LIN {X 0,Y 168.343,Z 1185.005,A -85,B 0,C 180,E1 2241.805,E2 2241.805} C_VEL
LIN {X 0,Y 169.597,Z 1183.384,A -85,B 0,C 180,E1 2234.616,E2 2234.616} C_VEL
LIN {X 0,Y 172.473,Z 1180.747,A -85,B 0,C 180,E1 2227.505,E2 2227.505} C_VEL
LIN {X 0,Y 177.252,Z 1177.063,A -85,B 0,C 180,E1 2220.61,E2 2220.61} C_VEL
LIN {X 0,Y 185.536,Z 1171.322,A -85,B 0,C 180,E1 2212.874,E2 2212.874} C_VEL
LIN {X 0,Y 197.006,Z 1163.471,A -85,B 0,C 180,E1 2205.542,E2 2205.542} C_VEL
LIN {X 0,Y 208.194,Z 1155.807,A -85,B 0,C 180,E1 2200.217,E2 2200.217} C_VEL
LIN {X 0,Y 221.519,Z 1146.423,A -85,B 0,C 180,E1 2195.217,E2 2195.217} C_VEL
LIN {X 0,Y 239.062,Z 1133.277,A -85,B 0,C 180,E1 2190.029,E2 2190.029} C_VEL
LIN {X 0,Y 253.681,Z 1121.544,A -85,B 0,C 180,E1 2186.529,E2 2186.529} C_VEL
LIN {X 0,Y 268.978,Z 1108.424,A -85,B 0,C 180,E1 2183.438,E2 2183.438} C_VEL
LIN {X 0,Y 287.731,Z 1090.816,A -85,B 0,C 180,E1 2180.24,E2 2180.24} C_VEL
LIN {X 0,Y 302.104,Z 1076.015,A -85,B 0,C 180,E1 2178.127,E2 2178.127} C_VEL
LIN {X 0,Y 316.159,Z 1060.322,A -85,B 0,C 180,E1 2176.294,E2 2176.294} C_VEL
LIN {X 0,Y 332.424,Z 1040.407,A -85,B 0,C 180,E1 2174.415,E2 2174.415} C_VEL
LIN {X 0,Y 346.747,Z 1020.63,A -85,B 0,C 180,E1 2172.929,E2 2172.929} C_VEL
LIN {X 0,Y 358.555,Z 1002.66,A -85,B 0,C 180,E1 2171.818,E2 2171.818} C_VEL
LIN {X 0,Y 370.024,Z 983.317,A -85,B 0,C 180,E1 2170.814,E2 2170.814} C_VEL
LIN {X 0,Y 383.165,Z 957.986,A -85,B 0,C 180,E1 2169.75,E2 2169.75} C_VEL
LIN {X 0,Y 392.344,Z 937.557,A -85,B 0,C 180,E1 2169.059,E2 2169.059} C_VEL
LIN {X 0,Y 400.34,Z 917.228,A -85,B 0,C 180,E1 2168.494,E2 2168.494} C_VEL
LIN {X 0,Y 408.607,Z 892.645,A -85,B 0,C 180,E1 2167.932,E2 2167.932} C_VEL
LIN {X 0,Y 415.555,Z 866.383,A -85,B 0,C 180,E1 2167.476,E2 2167.476} C_VEL
LIN {X 0,Y 420.191,Z 844.048,A -85,B 0,C 180,E1 2167.159,E2 2167.159} C_VEL
LIN {X 0,Y 424.177,Z 817.755,A -85,B 0,C 180,E1 2166.815,E2 2166.815} C_VEL
LIN {X 0,Y 442.106,Z 663.834,A -85,B 0,C 180,E1 2164.898,E2 2164.898} C_VEL
LIN {X 0,Y 441.771,Z 661.822,A -85,B 0,C 180,E1 2162.724,E2 2162.724} C_VEL
LIN {X 0,Y 442.134,Z 661.954,A -85,B 0,C 180,E1 2159.482,E2 2159.482} C_VEL
LIN {X 0,Y 442.426,Z 662.695,A -85,B 0,C 180,E1 2158.54,E2 2158.54} C_VEL
LIN {X 0,Y 440.538,Z 678.75,A -85,B 0,C 180,E1 2158.335,E2 2158.335} C_VEL
LIN {X 0,Y 439.566,Z 686.453,A -85,B 0,C 180,E1 2158.372,E2 2158.372} C_VEL
LIN {X 0,Y 436.764,Z 707.079,A -85,B 0,C 180,E1 2158.925,E2 2158.925} C_VEL
LIN {X 0,Y 435.94,Z 713.684,A -85,B 0,C 180,E1 2158.942,E2 2158.942} C_VEL
LIN {X 0,Y 422.165,Z 828.688,A -85,B 0,C 180,E1 2157.483,E2 2157.483} C_VEL
LIN {X 0,Y 417.336,Z 856.018,A -85,B 0,C 180,E1 2157.112,E2 2157.112} C_VEL
LIN {X 0,Y 411.12,Z 881.201,A -85,B 0,C 180,E1 2156.722,E2 2156.722} C_VEL
LIN {X 0,Y 404.786,Z 902.207,A -85,B 0,C 180,E1 2156.312,E2 2156.312} C_VEL
LIN {X 0,Y 397.021,Z 924.035,A -85,B 0,C 180,E1 2155.787,E2 2155.787} C_VEL
LIN {X 0,Y 385.817,Z 950.494,A -85,B 0,C 180,E1 2154.997,E2 2154.997} C_VEL
LIN {X 0,Y 375.845,Z 970.771,A -85,B 0,C 180,E1 2154.247,E2 2154.247} C_VEL
LIN {X 0,Y 364.942,Z 990.522,A -85,B 0,C 180,E1 2153.372,E2 2153.372} C_VEL
LIN {X 0,Y 350.842,Z 1013.342,A -85,B 0,C 180,E1 2152.137,E2 2152.137} C_VEL
LIN {X 0,Y 336.327,Z 1033.918,A -85,B 0,C 180,E1 2150.753,E2 2150.753} C_VEL
LIN {X 0,Y 323.015,Z 1051.093,A -85,B 0,C 180,E1 2149.357,E2 2149.357} C_VEL
LIN {X 0,Y 308.128,Z 1068.687,A -85,B 0,C 180,E1 2147.617,E2 2147.617} C_VEL
LIN {X 0,Y 289.64,Z 1088.449,A -85,B 0,C 180,E1 2145.148,E2 2145.148} C_VEL
LIN {X 0,Y 274.268,Z 1103.426,A -85,B 0,C 180,E1 2142.774,E2 2142.774} C_VEL
LIN {X 0,Y 259.412,Z 1116.892,A -85,B 0,C 180,E1 2140.13,E2 2140.13} C_VEL
LIN {X 0,Y 241.293,Z 1132.218,A -85,B 0,C 180,E1 2136.299,E2 2136.299} C_VEL
LIN {X 0,Y 224.396,Z 1145.324,A -85,B 0,C 180,E1 2131.915,E2 2131.915} C_VEL
LIN {X 0,Y 210.851,Z 1155.366,A -85,B 0,C 180,E1 2127.574,E2 2127.574} C_VEL
LIN {X 0,Y 197.418,Z 1165.01,A -85,B 0,C 180,E1 2122.194,E2 2122.194} C_VEL
LIN {X 0,Y 183.406,Z 1174.86,A -85,B 0,C 180,E1 2114.689,E2 2114.689} C_VEL
LIN {X 0,Y 174.298,Z 1181.394,A -85,B 0,C 180,E1 2107.865,E2 2107.865} C_VEL
LIN {X 0,Y 167.735,Z 1186.474,A -85,B 0,C 180,E1 2100.84,E2 2100.84} C_VEL
LIN {X 0,Y 163.294,Z 1190.442,A -85,B 0,C 180,E1 2093.453,E2 2093.453} C_VEL
LIN {X 0,Y 160.718,Z 1193.56,A -85,B 0,C 180,E1 2085.146,E2 2085.146} C_VEL
LIN {X 0,Y 160.036,Z 1195.327,A -85,B 0,C 180,E1 2077.177,E2 2077.177} C_VEL
LIN {X 0,Y 160.041,Z 1195.799,A -85,B 0,C 180,E1 2070.715,E2 2070.715} C_VEL
LIN {X 0,Y 160.019,Z 1195.475,A -85,B 0,C 180,E1 2064.621,E2 2064.621} C_VEL
LIN {X 0,Y 160.309,Z 1194.285,A -85,B 0,C 180,E1 2057.756,E2 2057.756} C_VEL
LIN {X 0,Y 162.268,Z 1191.586,A -85,B 0,C 180,E1 2049.059,E2 2049.059} C_VEL
LIN {X 0,Y 166.971,Z 1187.087,A -85,B 0,C 180,E1 2040.195,E2 2040.195} C_VEL
LIN {X 0,Y 173.231,Z 1182.143,A -85,B 0,C 180,E1 2033.109,E2 2033.109} C_VEL
LIN {X 0,Y 181.58,Z 1176.06,A -85,B 0,C 180,E1 2026.502,E2 2026.502} C_VEL
LIN {X 0,Y 192.698,Z 1168.241,A -85,B 0,C 180,E1 2020.048,E2 2020.048} C_VEL
LIN {X 0,Y 208.924,Z 1156.69,A -85,B 0,C 180,E1 2013.12,E2 2013.12} C_VEL
LIN {X 0,Y 222.987,Z 1146.275,A -85,B 0,C 180,E1 2008.493,E2 2008.493} C_VEL
LIN {X 0,Y 237.523,Z 1135.019,A -85,B 0,C 180,E1 2004.593,E2 2004.593} C_VEL
LIN {X 0,Y 256.179,Z 1119.593,A -85,B 0,C 180,E1 2000.489,E2 2000.489} C_VEL
LIN {X 0,Y 272.582,Z 1104.81,A -85,B 0,C 180,E1 1997.497,E2 1997.497} C_VEL
LIN {X 0,Y 287.038,Z 1090.825,A -85,B 0,C 180,E1 1995.222,E2 1995.222} C_VEL
LIN {X 0,Y 303.678,Z 1073.442,A -85,B 0,C 180,E1 1992.938,E2 1992.938} C_VEL
LIN {X 0,Y 321.192,Z 1053.061,A -85,B 0,C 180,E1 1990.837,E2 1990.837} C_VEL
LIN {X 0,Y 334.475,Z 1036.062,A -85,B 0,C 180,E1 1989.424,E2 1989.424} C_VEL
LIN {X 0,Y 346.809,Z 1018.795,A -85,B 0,C 180,E1 1988.215,E2 1988.215} C_VEL
LIN {X 0,Y 361.151,Z 996.648,A -85,B 0,C 180,E1 1986.94,E2 1986.94} C_VEL
LIN {X 0,Y 373.931,Z 973.923,A -85,B 0,C 180,E1 1985.892,E2 1985.892} C_VEL
LIN {X 0,Y 383.509,Z 954.818,A -85,B 0,C 180,E1 1985.16,E2 1985.16} C_VEL
LIN {X 0,Y 392.18,Z 935.339,A -85,B 0,C 180,E1 1984.533,E2 1984.533} C_VEL
LIN {X 0,Y 401.871,Z 910.318,A -85,B 0,C 180,E1 1983.875,E2 1983.875} C_VEL
LIN {X 0,Y 409.874,Z 884.69,A -85,B 0,C 180,E1 1983.344,E2 1983.344} C_VEL
LIN {X 0,Y 415.471,Z 862.848,A -85,B 0,C 180,E1 1982.989,E2 1982.989} C_VEL
LIN {X 0,Y 420.46,Z 838.069,A -85,B 0,C 180,E1 1982.645,E2 1982.645} C_VEL
LIN {X 0,Y 425.272,Z 801.988,A -85,B 0,C 180,E1 1982.176,E2 1982.176} C_VEL
LIN {X 0,Y 440.907,Z 669.688,A -85,B 0,C 180,E1 1980.487,E2 1980.487} C_VEL
LIN {X 0,Y 440.543,Z 669.536,A -85,B 0,C 180,E1 1977.268,E2 1977.268} C_VEL
LIN {X 0,Y 440.641,Z 670.612,A -85,B 0,C 180,E1 1975.958,E2 1975.958} C_VEL
LIN {X 0,Y 421.733,Z 828.746,A -85,B 0,C 180,E1 1974.036,E2 1974.036} C_VEL
LIN {X 0,Y 417.043,Z 855.632,A -85,B 0,C 180,E1 1973.685,E2 1973.685} C_VEL
LIN {X 0,Y 410.82,Z 880.969,A -85,B 0,C 180,E1 1973.3,E2 1973.3} C_VEL
LIN {X 0,Y 404.54,Z 901.829,A -85,B 0,C 180,E1 1972.915,E2 1972.915} C_VEL
LIN {X 0,Y 396.455,Z 924.553,A -85,B 0,C 180,E1 1972.379,E2 1972.379} C_VEL
LIN {X 0,Y 385.571,Z 950.141,A -85,B 0,C 180,E1 1971.621,E2 1971.621} C_VEL
LIN {X 0,Y 375.692,Z 970.166,A -85,B 0,C 180,E1 1970.893,E2 1970.893} C_VEL
LIN {X 0,Y 364.998,Z 989.466,A -85,B 0,C 180,E1 1970.049,E2 1970.049} C_VEL
LIN {X 0,Y 351.084,Z 1011.894,A -85,B 0,C 180,E1 1968.851,E2 1968.851} C_VEL
LIN {X 0,Y 336.43,Z 1032.521,A -85,B 0,C 180,E1 1967.469,E2 1967.469} C_VEL
LIN {X 0,Y 323.858,Z 1048.616,A -85,B 0,C 180,E1 1966.165,E2 1966.165} C_VEL
LIN {X 0,Y 310.107,Z 1064.74,A -85,B 0,C 180,E1 1964.595,E2 1964.595} C_VEL
LIN {X 0,Y 292.228,Z 1083.793,A -85,B 0,C 180,E1 1962.27,E2 1962.27} C_VEL
LIN {X 0,Y 275.903,Z 1099.429,A -85,B 0,C 180,E1 1959.822,E2 1959.822} C_VEL
LIN {X 0,Y 261.243,Z 1112.417,A -85,B 0,C 180,E1 1957.281,E2 1957.281} C_VEL
LIN {X 0,Y 243.843,Z 1126.755,A -85,B 0,C 180,E1 1953.713,E2 1953.713} C_VEL
LIN {X 0,Y 226.55,Z 1139.657,A -85,B 0,C 180,E1 1949.389,E2 1949.389} C_VEL
LIN {X 0,Y 213.03,Z 1149.178,A -85,B 0,C 180,E1 1945.224,E2 1945.224} C_VEL
LIN {X 0,Y 198.965,Z 1158.65,A -85,B 0,C 180,E1 1939.806,E2 1939.806} C_VEL
LIN {X 0,Y 185.194,Z 1167.496,A -85,B 0,C 180,E1 1932.753,E2 1932.753} C_VEL
LIN {X 0,Y 175.872,Z 1173.471,A -85,B 0,C 180,E1 1926.165,E2 1926.165} C_VEL
LIN {X 0,Y 168.774,Z 1178.214,A -85,B 0,C 180,E1 1919.066,E2 1919.066} C_VEL
LIN {X 0,Y 163.243,Z 1182.407,A -85,B 0,C 180,E1 1910.061,E2 1910.061} C_VEL
LIN {X 0,Y 160.765,Z 1184.715,A -85,B 0,C 180,E1 1901.481,E2 1901.481} C_VEL
LIN {X 0,Y 160.13,Z 1185.67,A -85,B 0,C 180,E1 1894.657,E2 1894.657} C_VEL
LIN {X 0,Y 160.081,Z 1185.848,A -85,B 0,C 180,E1 1888.211,E2 1888.211} C_VEL
LIN {X 0,Y 160.385,Z 1185.254,A -85,B 0,C 180,E1 1881.396,E2 1881.396} C_VEL
LIN {X 0,Y 161.788,Z 1183.633,A -85,B 0,C 180,E1 1873.853,E2 1873.853} C_VEL
LIN {X 0,Y 164.953,Z 1180.999,A -85,B 0,C 180,E1 1866.419,E2 1866.419} C_VEL
LIN {X 0,Y 170.141,Z 1177.318,A -85,B 0,C 180,E1 1859.252,E2 1859.252} C_VEL
LIN {X 0,Y 179.028,Z 1171.576,A -85,B 0,C 180,E1 1851.28,E2 1851.28} C_VEL
LIN {X 0,Y 191.191,Z 1163.728,A -85,B 0,C 180,E1 1843.806,E2 1843.806} C_VEL
LIN {X 0,Y 202.953,Z 1156.065,A -85,B 0,C 180,E1 1838.434,E2 1838.434} C_VEL
LIN {X 0,Y 216.854,Z 1146.684,A -85,B 0,C 180,E1 1833.431,E2 1833.431} C_VEL
LIN {X 0,Y 235.038,Z 1133.544,A -85,B 0,C 180,E1 1828.286,E2 1828.286} C_VEL
LIN {X 0,Y 250.303,Z 1121.658,A -85,B 0,C 180,E1 1824.8,E2 1824.8} C_VEL
LIN {X 0,Y 265.964,Z 1108.571,A -85,B 0,C 180,E1 1821.786,E2 1821.786} C_VEL
LIN {X 0,Y 285,Z 1091.104,A -85,B 0,C 180,E1 1818.694,E2 1818.694} C_VEL
LIN {X 0,Y 299.534,Z 1076.446,A -85,B 0,C 180,E1 1816.659,E2 1816.659} C_VEL
LIN {X 0,Y 313.528,Z 1061.128,A -85,B 0,C 180,E1 1814.918,E2 1814.918} C_VEL
LIN {X 0,Y 330.046,Z 1041.343,A -85,B 0,C 180,E1 1813.099,E2 1813.099} C_VEL
LIN {X 0,Y 345.026,Z 1020.985,A -85,B 0,C 180,E1 1811.619,E2 1811.619} C_VEL
LIN {X 0,Y 356.989,Z 1003.038,A -85,B 0,C 180,E1 1810.55,E2 1810.55} C_VEL
LIN {X 0,Y 368.6,Z 983.725,A -85,B 0,C 180,E1 1809.586,E2 1809.586} C_VEL
LIN {X 0,Y 381.72,Z 958.832,A -85,B 0,C 180,E1 1808.577,E2 1808.577} C_VEL
LIN {X 0,Y 391.164,Z 938.102,A -85,B 0,C 180,E1 1807.902,E2 1807.902} C_VEL
LIN {X 0,Y 398.763,Z 919.118,A -85,B 0,C 180,E1 1807.392,E2 1807.392} C_VEL
LIN {X 0,Y 406.146,Z 897.763,A -85,B 0,C 180,E1 1806.907,E2 1806.907} C_VEL
LIN {X 0,Y 413.926,Z 870.284,A -85,B 0,C 180,E1 1806.43,E2 1806.43} C_VEL
LIN {X 0,Y 419.128,Z 846.122,A -85,B 0,C 180,E1 1806.096,E2 1806.096} C_VEL
LIN {X 0,Y 422.769,Z 823.388,A -85,B 0,C 180,E1 1805.803,E2 1805.803} C_VEL
LIN {X 0,Y 440.908,Z 670.849,A -85,B 0,C 180,E1 1803.934,E2 1803.934} C_VEL
LIN {X 0,Y 440.785,Z 669.741,A -85,B 0,C 180,E1 1802.6,E2 1802.6} C_VEL
LIN {X 0,Y 441.146,Z 669.924,A -85,B 0,C 180,E1 1799.489,E2 1799.489} C_VEL
LIN {X 0,Y 435.94,Z 713.684,A -85,B 0,C 180,E1 1798.942,E2 1798.942} C_VEL
LIN {X 0,Y 434.973,Z 721.387,A -85,B 0,C 180,E1 1798.978,E2 1798.978} C_VEL
LIN {X 0,Y 432.22,Z 742.01,A -85,B 0,C 180,E1 1799.55,E2 1799.55} C_VEL
LIN {X 0,Y 431.4,Z 748.617,A -85,B 0,C 180,E1 1799.567,E2 1799.567} C_VEL
LIN {X 0,Y 421.531,Z 829.434,A -85,B 0,C 180,E1 1798.562,E2 1798.562} C_VEL
LIN {X 0,Y 416.387,Z 857.626,A -85,B 0,C 180,E1 1798.19,E2 1798.19} C_VEL
LIN {X 0,Y 410.366,Z 881.665,A -85,B 0,C 180,E1 1797.832,E2 1797.832} C_VEL
LIN {X 0,Y 403.902,Z 902.829,A -85,B 0,C 180,E1 1797.435,E2 1797.435} C_VEL
LIN {X 0,Y 395.04,Z 927.3,A -85,B 0,C 180,E1 1796.865,E2 1796.865} C_VEL
LIN {X 0,Y 384.318,Z 951.817,A -85,B 0,C 180,E1 1796.15,E2 1796.15} C_VEL
LIN {X 0,Y 374.707,Z 971.077,A -85,B 0,C 180,E1 1795.465,E2 1795.465} C_VEL
LIN {X 0,Y 363.825,Z 990.545,A -85,B 0,C 180,E1 1794.638,E2 1794.638} C_VEL
LIN {X 0,Y 349.723,Z 1013.098,A -85,B 0,C 180,E1 1793.47,E2 1793.47} C_VEL
LIN {X 0,Y 335.093,Z 1033.573,A -85,B 0,C 180,E1 1792.155,E2 1792.155} C_VEL
LIN {X 0,Y 321.581,Z 1050.765,A -85,B 0,C 180,E1 1790.816,E2 1790.816} C_VEL
LIN {X 0,Y 307.001,Z 1067.746,A -85,B 0,C 180,E1 1789.206,E2 1789.206} C_VEL
LIN {X 0,Y 287.606,Z 1088.154,A -85,B 0,C 180,E1 1786.762,E2 1786.762} C_VEL
LIN {X 0,Y 271.899,Z 1103.136,A -85,B 0,C 180,E1 1784.465,E2 1784.465} C_VEL
LIN {X 0,Y 256.672,Z 1116.609,A -85,B 0,C 180,E1 1781.898,E2 1781.898} C_VEL
LIN {X 0,Y 238.046,Z 1131.929,A -85,B 0,C 180,E1 1778.166,E2 1778.166} C_VEL
LIN {X 0,Y 220.537,Z 1145.053,A -85,B 0,C 180,E1 1773.855,E2 1773.855} C_VEL
LIN {X 0,Y 206.433,Z 1155.098,A -85,B 0,C 180,E1 1769.559,E2 1769.559} C_VEL
LIN {X 0,Y 192.353,Z 1164.745,A -85,B 0,C 180,E1 1764.184,E2 1764.184} C_VEL
LIN {X 0,Y 177.473,Z 1174.624,A -85,B 0,C 180,E1 1756.579,E2 1756.579} C_VEL
LIN {X 0,Y 167.755,Z 1181.135,A -85,B 0,C 180,E1 1749.624,E2 1749.624} C_VEL
LIN {X 0,Y 160.635,Z 1186.217,A -85,B 0,C 180,E1 1742.364,E2 1742.364} C_VEL
LIN {X 0,Y 155.743,Z 1190.187,A -85,B 0,C 180,E1 1734.663,E2 1734.663} C_VEL
LIN {X 0,Y 152.847,Z 1193.316,A -85,B 0,C 180,E1 1725.92,E2 1725.92} C_VEL
LIN {X 0,Y 152.051,Z 1195.078,A -85,B 0,C 180,E1 1717.557,E2 1717.557} C_VEL
LIN {X 0,Y 152.045,Z 1195.552,A -85,B 0,C 180,E1 1710.753,E2 1710.753} C_VEL
LIN {X 0,Y 152.022,Z 1195.227,A -85,B 0,C 180,E1 1704.337,E2 1704.337} C_VEL
LIN {X 0,Y 152.373,Z 1194.034,A -85,B 0,C 180,E1 1697.107,E2 1697.107} C_VEL
LIN {X 0,Y 154.6,Z 1191.33,A -85,B 0,C 180,E1 1687.968,E2 1687.968} C_VEL
LIN {X 0,Y 159.801,Z 1186.827,A -85,B 0,C 180,E1 1678.712,E2 1678.712} C_VEL
LIN {X 0,Y 166.815,Z 1181.732,A -85,B 0,C 180,E1 1671.19,E2 1671.19} C_VEL
LIN {X 0,Y 176.024,Z 1175.499,A -85,B 0,C 180,E1 1664.322,E2 1664.322} C_VEL
LIN {X 0,Y 189.382,Z 1166.704,A -85,B 0,C 180,E1 1657.132,E2 1657.132} C_VEL
LIN {X 0,Y 205.086,Z 1155.945,A -85,B 0,C 180,E1 1650.898,E2 1650.898} C_VEL
LIN {X 0,Y 219.073,Z 1146.002,A -85,B 0,C 180,E1 1646.546,E2 1646.546} C_VEL
LIN {X 0,Y 234.127,Z 1134.74,A -85,B 0,C 180,E1 1642.71,E2 1642.71} C_VEL
LIN {X 0,Y 253.351,Z 1119.304,A -85,B 0,C 180,E1 1638.703,E2 1638.703} C_VEL
LIN {X 0,Y 270.173,Z 1104.518,A -85,B 0,C 180,E1 1635.797,E2 1635.797} C_VEL
LIN {X 0,Y 284.949,Z 1090.524,A -85,B 0,C 180,E1 1633.593,E2 1633.593} C_VEL
LIN {X 0,Y 302.817,Z 1072.194,A -85,B 0,C 180,E1 1631.282,E2 1631.282} C_VEL
LIN {X 0,Y 319.867,Z 1052.554,A -85,B 0,C 180,E1 1629.355,E2 1629.355} C_VEL
LIN {X 0,Y 333.216,Z 1035.707,A -85,B 0,C 180,E1 1628.015,E2 1628.015} C_VEL
LIN {X 0,Y 345.923,Z 1018.139,A -85,B 0,C 180,E1 1626.842,E2 1626.842} C_VEL
LIN {X 0,Y 360.68,Z 995.478,A -85,B 0,C 180,E1 1625.602,E2 1625.602} C_VEL
LIN {X 0,Y 373.177,Z 973.455,A -85,B 0,C 180,E1 1624.637,E2 1624.637} C_VEL
LIN {X 0,Y 382.859,Z 954.303,A -85,B 0,C 180,E1 1623.939,E2 1623.939} C_VEL
LIN {X 0,Y 392.093,Z 933.656,A -85,B 0,C 180,E1 1623.31,E2 1623.31} C_VEL
LIN {X 0,Y 402.382,Z 906.609,A -85,B 0,C 180,E1 1622.65,E2 1622.65} C_VEL
LIN {X 0,Y 409.535,Z 883.617,A -85,B 0,C 180,E1 1622.205,E2 1622.205} C_VEL
LIN {X 0,Y 415.13,Z 861.776,A -85,B 0,C 180,E1 1621.869,E2 1621.869} C_VEL
LIN {X 0,Y 420.483,Z 834.821,A -85,B 0,C 180,E1 1621.51,E2 1621.51} C_VEL
LIN {X 0,Y 426.138,Z 790.486,A -85,B 0,C 180,E1 1620.954,E2 1620.954} C_VEL
LIN {X 0,Y 439.703,Z 677.389,A -85,B 0,C 180,E1 1619.544,E2 1619.544} C_VEL
LIN {X 0,Y 439.583,Z 677.674,A -85,B 0,C 180,E1 1616.92,E2 1616.92} C_VEL
LIN {X 0,Y 421.221,Z 828.841,A -85,B 0,C 180,E1 1615.124,E2 1615.124} C_VEL
LIN {X 0,Y 416.416,Z 855.943,A -85,B 0,C 180,E1 1614.782,E2 1614.782} C_VEL
LIN {X 0,Y 410.209,Z 880.97,A -85,B 0,C 180,E1 1614.418,E2 1614.418} C_VEL
LIN {X 0,Y 403.876,Z 901.826,A -85,B 0,C 180,E1 1614.053,E2 1614.053} C_VEL
LIN {X 0,Y 395.955,Z 923.911,A -85,B 0,C 180,E1 1613.555,E2 1613.555} C_VEL
LIN {X 0,Y 384.963,Z 949.648,A -85,B 0,C 180,E1 1612.833,E2 1612.833} C_VEL
LIN {X 0,Y 374.978,Z 969.731,A -85,B 0,C 180,E1 1612.141,E2 1612.141} C_VEL
LIN {X 0,Y 364.117,Z 989.163,A -85,B 0,C 180,E1 1611.331,E2 1611.331} C_VEL
LIN {X 0,Y 350.546,Z 1010.866,A -85,B 0,C 180,E1 1610.228,E2 1610.228} C_VEL
LIN {X 0,Y 335.267,Z 1032.21,A -85,B 0,C 180,E1 1608.87,E2 1608.87} C_VEL
LIN {X 0,Y 322.011,Z 1048.944,A -85,B 0,C 180,E1 1607.571,E2 1607.571} C_VEL
LIN {X 0,Y 307.595,Z 1065.554,A -85,B 0,C 180,E1 1606.005,E2 1606.005} C_VEL
LIN {X 0,Y 288.638,Z 1085.236,A -85,B 0,C 180,E1 1603.652,E2 1603.652} C_VEL
LIN {X 0,Y 273.108,Z 1099.782,A -85,B 0,C 180,E1 1601.426,E2 1601.426} C_VEL
LIN {X 0,Y 258.178,Z 1112.698,A -85,B 0,C 180,E1 1598.964,E2 1598.964} C_VEL
LIN {X 0,Y 239.796,Z 1127.407,A -85,B 0,C 180,E1 1595.368,E2 1595.368} C_VEL
LIN {X 0,Y 222.455,Z 1139.922,A -85,B 0,C 180,E1 1591.221,E2 1591.221} C_VEL
LIN {X 0,Y 208.423,Z 1149.44,A -85,B 0,C 180,E1 1587.092,E2 1587.092} C_VEL
LIN {X 0,Y 193.731,Z 1158.911,A -85,B 0,C 180,E1 1581.675,E2 1581.675} C_VEL
LIN {X 0,Y 179.355,Z 1167.675,A -85,B 0,C 180,E1 1574.623,E2 1574.623} C_VEL
LIN {X 0,Y 169.371,Z 1173.678,A -85,B 0,C 180,E1 1567.877,E2 1567.877} C_VEL
LIN {X 0,Y 161.651,Z 1178.469,A -85,B 0,C 180,E1 1560.479,E2 1560.479} C_VEL
LIN {X 0,Y 155.611,Z 1182.658,A -85,B 0,C 180,E1 1551.09,E2 1551.09} C_VEL
LIN {X 0,Y 152.855,Z 1184.965,A -85,B 0,C 180,E1 1542.083,E2 1542.083} C_VEL
LIN {X 0,Y 152.143,Z 1185.918,A -85,B 0,C 180,E1 1534.902,E2 1534.902} C_VEL
LIN {X 0,Y 152.084,Z 1186.117,A -85,B 0,C 180,E1 1528.494,E2 1528.494} C_VEL
LIN {X 0,Y 152.428,Z 1185.502,A -85,B 0,C 180,E1 1520.943,E2 1520.943} C_VEL
LIN {X 0,Y 154.007,Z 1183.884,A -85,B 0,C 180,E1 1513.014,E2 1513.014} C_VEL
LIN {X 0,Y 157.503,Z 1181.242,A -85,B 0,C 180,E1 1505.207,E2 1505.207} C_VEL
LIN {X 0,Y 163.453,Z 1177.373,A -85,B 0,C 180,E1 1497.432,E2 1497.432} C_VEL
LIN {X 0,Y 173.561,Z 1171.317,A -85,B 0,C 180,E1 1488.949,E2 1488.949} C_VEL
LIN {X 0,Y 186.115,Z 1163.643,A -85,B 0,C 180,E1 1481.691,E2 1481.691} C_VEL
LIN {X 0,Y 198.543,Z 1155.931,A -85,B 0,C 180,E1 1476.316,E2 1476.316} C_VEL
LIN {X 0,Y 214.497,Z 1145.598,A -85,B 0,C 180,E1 1470.94,E2 1470.94} C_VEL
LIN {X 0,Y 231.997,Z 1133.25,A -85,B 0,C 180,E1 1466.306,E2 1466.306} C_VEL
LIN {X 0,Y 246.762,Z 1122.082,A -85,B 0,C 180,E1 1463.104,E2 1463.104} C_VEL
LIN {X 0,Y 262.194,Z 1109.532,A -85,B 0,C 180,E1 1460.263,E2 1460.263} C_VEL
LIN {X 0,Y 281.621,Z 1092.223,A -85,B 0,C 180,E1 1457.242,E2 1457.242} C_VEL
LIN {X 0,Y 297.296,Z 1076.74,A -85,B 0,C 180,E1 1455.151,E2 1455.151} C_VEL
LIN {X 0,Y 311.531,Z 1061.433,A -85,B 0,C 180,E1 1453.471,E2 1453.471} C_VEL
LIN {X 0,Y 328.302,Z 1041.673,A -85,B 0,C 180,E1 1451.719,E2 1451.719} C_VEL
LIN {X 0,Y 343.487,Z 1021.339,A -85,B 0,C 180,E1 1450.296,E2 1450.296} C_VEL
LIN {X 0,Y 355.6,Z 1003.417,A -85,B 0,C 180,E1 1449.271,E2 1449.271} C_VEL
LIN {X 0,Y 366.873,Z 984.936,A -85,B 0,C 180,E1 1448.384,E2 1448.384} C_VEL
LIN {X 0,Y 379.657,Z 961.31,A -85,B 0,C 180,E1 1447.452,E2 1447.452} C_VEL
LIN {X 0,Y 390.144,Z 938.645,A -85,B 0,C 180,E1 1446.738,E2 1446.738} C_VEL
LIN {X 0,Y 398.295,Z 918.46,A -85,B 0,C 180,E1 1446.222,E2 1446.222} C_VEL
LIN {X 0,Y 405.748,Z 897.006,A -85,B 0,C 180,E1 1445.762,E2 1445.762} C_VEL
LIN {X 0,Y 413.83,Z 868.219,A -85,B 0,C 180,E1 1445.291,E2 1445.291} C_VEL
LIN {X 0,Y 418.752,Z 845.309,A -85,B 0,C 180,E1 1444.989,E2 1444.989} C_VEL
LIN {X 0,Y 422.461,Z 822.137,A -85,B 0,C 180,E1 1444.702,E2 1444.702} C_VEL
LIN {X 0,Y 439.837,Z 677.848,A -85,B 0,C 180,E1 1442.965,E2 1442.965} C_VEL
LIN {X 0,Y 439.934,Z 677.599,A -85,B 0,C 180,E1 1440.44,E2 1440.44} C_VEL
LIN {X 0,Y 431.4,Z 748.617,A -85,B 0,C 180,E1 1439.567,E2 1439.567} C_VEL
LIN {X 0,Y 430.444,Z 756.318,A -85,B 0,C 180,E1 1439.603,E2 1439.603} C_VEL
LIN {X 0,Y 427.764,Z 776.936,A -85,B 0,C 180,E1 1440.189,E2 1440.189} C_VEL
LIN {X 0,Y 426.948,Z 783.545,A -85,B 0,C 180,E1 1440.211,E2 1440.211} C_VEL
LIN {X 0,Y 420.687,Z 832.7,A -85,B 0,C 180,E1 1439.612,E2 1439.612} C_VEL
LIN {X 0,Y 415.232,Z 860.734,A -85,B 0,C 180,E1 1439.253,E2 1439.253} C_VEL
LIN {X 0,Y 409.511,Z 883.03,A -85,B 0,C 180,E1 1438.931,E2 1438.931} C_VEL
LIN {X 0,Y 402.581,Z 905.247,A -85,B 0,C 180,E1 1438.528,E2 1438.528} C_VEL
LIN {X 0,Y 392.213,Z 932.569,A -85,B 0,C 180,E1 1437.9,E2 1437.9} C_VEL
LIN {X 0,Y 382.882,Z 953.332,A -85,B 0,C 180,E1 1437.306,E2 1437.306} C_VEL
LIN {X 0,Y 372.604,Z 973.503,A -85,B 0,C 180,E1 1436.61,E2 1436.61} C_VEL
LIN {X 0,Y 359.487,Z 996.336,A -85,B 0,C 180,E1 1435.654,E2 1435.654} C_VEL
LIN {X 0,Y 344.559,Z 1018.824,A -85,B 0,C 180,E1 1434.47,E2 1434.47} C_VEL
LIN {X 0,Y 331.689,Z 1036.313,A -85,B 0,C 180,E1 1433.349,E2 1433.349} C_VEL
LIN {X 0,Y 316.706,Z 1054.829,A -85,B 0,C 180,E1 1431.917,E2 1431.917} C_VEL
LIN {X 0,Y 298.081,Z 1075.425,A -85,B 0,C 180,E1 1429.9,E2 1429.9} C_VEL
LIN {X 0,Y 282.202,Z 1091.304,A -85,B 0,C 180,E1 1427.93,E2 1427.93} C_VEL
LIN {X 0,Y 266.156,Z 1106.088,A -85,B 0,C 180,E1 1425.644,E2 1425.644} C_VEL
LIN {X 0,Y 245.732,Z 1123.238,A -85,B 0,C 180,E1 1422.2,E2 1422.2} C_VEL
LIN {X 0,Y 229.402,Z 1135.773,A -85,B 0,C 180,E1 1418.865,E2 1418.865} C_VEL
LIN {X 0,Y 213.924,Z 1146.9,A -85,B 0,C 180,E1 1415.059,E2 1415.059} C_VEL
LIN {X 0,Y 196.064,Z 1159.035,A -85,B 0,C 180,E1 1409.524,E2 1409.524} C_VEL
LIN {X 0,Y 180.766,Z 1168.723,A -85,B 0,C 180,E1 1403.316,E2 1403.316} C_VEL
LIN {X 0,Y 169.259,Z 1175.916,A -85,B 0,C 180,E1 1397.097,E2 1397.097} C_VEL
LIN {X 0,Y 159.335,Z 1182.205,A -85,B 0,C 180,E1 1389.797,E2 1389.797} C_VEL
LIN {X 0,Y 150.547,Z 1188.236,A -85,B 0,C 180,E1 1379.875,E2 1379.875} C_VEL
LIN {X 0,Y 145.983,Z 1191.961,A -85,B 0,C 180,E1 1370.444,E2 1370.444} C_VEL
LIN {X 0,Y 144.356,Z 1193.945,A -85,B 0,C 180,E1 1362.805,E2 1362.805} C_VEL
LIN {X 0,Y 144.027,Z 1195.009,A -85,B 0,C 180,E1 1355.577,E2 1355.577} C_VEL
LIN {X 0,Y 144.048,Z 1195.301,A -85,B 0,C 180,E1 1349.204,E2 1349.204} C_VEL
LIN {X 0,Y 144.054,Z 1194.872,A -85,B 0,C 180,E1 1342.421,E2 1342.421} C_VEL
LIN {X 0,Y 144.938,Z 1193.14,A -85,B 0,C 180,E1 1333.523,E2 1333.523} C_VEL
LIN {X 0,Y 148.065,Z 1190.067,A -85,B 0,C 180,E1 1324.392,E2 1324.392} C_VEL
LIN {X 0,Y 153.343,Z 1186.133,A -85,B 0,C 180,E1 1316.34,E2 1316.34} C_VEL
LIN {X 0,Y 160.959,Z 1181.088,A -85,B 0,C 180,E1 1308.816,E2 1308.816} C_VEL
LIN {X 0,Y 171.299,Z 1174.585,A -85,B 0,C 180,E1 1301.656,E2 1301.656} C_VEL
LIN {X 0,Y 186.895,Z 1164.805,A -85,B 0,C 180,E1 1293.978,E2 1293.978} C_VEL
LIN {X 0,Y 201.568,Z 1155.202,A -85,B 0,C 180,E1 1288.596,E2 1288.596} C_VEL
LIN {X 0,Y 216.344,Z 1145.084,A -85,B 0,C 180,E1 1284.289,E2 1284.289} C_VEL
LIN {X 0,Y 234.22,Z 1132.114,A -85,B 0,C 180,E1 1280.086,E2 1280.086} C_VEL
LIN {X 0,Y 253.324,Z 1116.87,A -85,B 0,C 180,E1 1276.436,E2 1276.436} C_VEL
LIN {X 0,Y 268.887,Z 1103.439,A -85,B 0,C 180,E1 1273.938,E2 1273.938} C_VEL
LIN {X 0,Y 284.897,Z 1088.5,A -85,B 0,C 180,E1 1271.71,E2 1271.71} C_VEL
LIN {X 0,Y 304.613,Z 1068.197,A -85,B 0,C 180,E1 1269.351,E2 1269.351} C_VEL
LIN {X 0,Y 319.416,Z 1051.257,A -85,B 0,C 180,E1 1267.797,E2 1267.797} C_VEL
LIN {X 0,Y 333.109,Z 1034.12,A -85,B 0,C 180,E1 1266.51,E2 1266.51} C_VEL
LIN {X 0,Y 348.398,Z 1013.029,A -85,B 0,C 180,E1 1265.21,E2 1265.21} C_VEL
LIN {X 0,Y 362.374,Z 990.968,A -85,B 0,C 180,E1 1264.114,E2 1264.114} C_VEL
LIN {X 0,Y 373.091,Z 972.076,A -85,B 0,C 180,E1 1263.343,E2 1263.343} C_VEL
LIN {X 0,Y 382.874,Z 952.774,A -85,B 0,C 180,E1 1262.683,E2 1262.683} C_VEL
LIN {X 0,Y 393.477,Z 928.982,A -85,B 0,C 180,E1 1262.013,E2 1262.013} C_VEL
LIN {X 0,Y 402.83,Z 903.623,A -85,B 0,C 180,E1 1261.444,E2 1261.444} C_VEL
LIN {X 0,Y 409.521,Z 881.976,A -85,B 0,C 180,E1 1261.055,E2 1261.055} C_VEL
LIN {X 0,Y 415.452,Z 858.564,A -85,B 0,C 180,E1 1260.72,E2 1260.72} C_VEL
LIN {X 0,Y 420.817,Z 829.737,A -85,B 0,C 180,E1 1260.353,E2 1260.353} C_VEL
LIN {X 0,Y 430.755,Z 749.544,A -85,B 0,C 180,E1 1259.379,E2 1259.379} C_VEL
LIN {X 0,Y 438.6,Z 685.248,A -85,B 0,C 180,E1 1258.599,E2 1258.599} C_VEL
LIN {X 0,Y 438.548,Z 685.499,A -85,B 0,C 180,E1 1257.877,E2 1257.877} C_VEL
LIN {X 0,Y 420.868,Z 828.891,A -85,B 0,C 180,E1 1256.215,E2 1256.215} C_VEL
LIN {X 0,Y 415.987,Z 856.065,A -85,B 0,C 180,E1 1255.884,E2 1255.884} C_VEL
LIN {X 0,Y 409.724,Z 881.081,A -85,B 0,C 180,E1 1255.538,E2 1255.538} C_VEL
LIN {X 0,Y 403.371,Z 901.823,A -85,B 0,C 180,E1 1255.193,E2 1255.193} C_VEL
LIN {X 0,Y 395.139,Z 924.544,A -85,B 0,C 180,E1 1254.705,E2 1254.705} C_VEL
LIN {X 0,Y 384.046,Z 950.149,A -85,B 0,C 180,E1 1254.019,E2 1254.019} C_VEL
LIN {X 0,Y 373.965,Z 970.187,A -85,B 0,C 180,E1 1253.36,E2 1253.36} C_VEL
LIN {X 0,Y 362.992,Z 989.582,A -85,B 0,C 180,E1 1252.587,E2 1252.587} C_VEL
LIN {X 0,Y 348.795,Z 1011.956,A -85,B 0,C 180,E1 1251.495,E2 1251.495} C_VEL
LIN {X 0,Y 333.797,Z 1032.554,A -85,B 0,C 180,E1 1250.235,E2 1250.235} C_VEL
LIN {X 0,Y 320.359,Z 1049.272,A -85,B 0,C 180,E1 1248.991,E2 1248.991} C_VEL
LIN {X 0,Y 304.956,Z 1066.719,A -85,B 0,C 180,E1 1247.403,E2 1247.403} C_VEL
LIN {X 0,Y 286.442,Z 1085.53,A -85,B 0,C 180,E1 1245.223,E2 1245.223} C_VEL
LIN {X 0,Y 270.682,Z 1100.002,A -85,B 0,C 180,E1 1243.084,E2 1243.084} C_VEL
LIN {X 0,Y 255.343,Z 1112.978,A -85,B 0,C 180,E1 1240.686,E2 1240.686} C_VEL
LIN {X 0,Y 236.478,Z 1127.675,A -85,B 0,C 180,E1 1237.184,E2 1237.184} C_VEL
LIN {X 0,Y 218.597,Z 1140.187,A -85,B 0,C 180,E1 1233.12,E2 1233.12} C_VEL
LIN {X 0,Y 203.994,Z 1149.738,A -85,B 0,C 180,E1 1229.025,E2 1229.025} C_VEL
LIN {X 0,Y 188.464,Z 1159.331,A -85,B 0,C 180,E1 1223.543,E2 1223.543} C_VEL
LIN {X 0,Y 173.574,Z 1167.931,A -85,B 0,C 180,E1 1216.539,E2 1216.539} C_VEL
LIN {X 0,Y 162.942,Z 1173.934,A -85,B 0,C 180,E1 1209.658,E2 1209.658} C_VEL
LIN {X 0,Y 154.632,Z 1178.725,A -85,B 0,C 180,E1 1202.022,E2 1202.022} C_VEL
LIN {X 0,Y 147.846,Z 1183.017,A -85,B 0,C 180,E1 1191.838,E2 1191.838} C_VEL
LIN {X 0,Y 144.959,Z 1185.214,A -85,B 0,C 180,E1 1182.752,E2 1182.752} C_VEL
LIN {X 0,Y 144.156,Z 1186.166,A -85,B 0,C 180,E1 1175.174,E2 1175.174} C_VEL
LIN {X 0,Y 144.088,Z 1186.364,A -85,B 0,C 180,E1 1168.41,E2 1168.41} C_VEL
LIN {X 0,Y 144.439,Z 1185.815,A -85,B 0,C 180,E1 1160.839,E2 1160.839} C_VEL
LIN {X 0,Y 146.258,Z 1184.135,A -85,B 0,C 180,E1 1152.084,E2 1152.084} C_VEL
LIN {X 0,Y 150.099,Z 1181.503,A -85,B 0,C 180,E1 1143.919,E2 1143.919} C_VEL
LIN {X 0,Y 156.583,Z 1177.626,A -85,B 0,C 180,E1 1135.811,E2 1135.811} C_VEL
LIN {X 0,Y 167.421,Z 1171.574,A -85,B 0,C 180,E1 1127.092,E2 1127.092} C_VEL
LIN {X 0,Y 180.721,Z 1163.9,A -85,B 0,C 180,E1 1119.733,E2 1119.733} C_VEL
LIN {X 0,Y 193.756,Z 1156.19,A -85,B 0,C 180,E1 1114.344,E2 1114.344} C_VEL
LIN {X 0,Y 209.639,Z 1146.305,A -85,B 0,C 180,E1 1109.213,E2 1109.213} C_VEL
LIN {X 0,Y 228.46,Z 1133.516,A -85,B 0,C 180,E1 1104.45,E2 1104.45} C_VEL
LIN {X 0,Y 243.647,Z 1122.349,A -85,B 0,C 180,E1 1101.322,E2 1101.322} C_VEL
LIN {X 0,Y 259.462,Z 1109.804,A -85,B 0,C 180,E1 1098.56,E2 1098.56} C_VEL
LIN {X 0,Y 278.426,Z 1093.341,A -85,B 0,C 180,E1 1095.756,E2 1095.756} C_VEL
LIN {X 0,Y 294.371,Z 1077.947,A -85,B 0,C 180,E1 1093.727,E2 1093.727} C_VEL
LIN {X 0,Y 308.822,Z 1062.739,A -85,B 0,C 180,E1 1092.101,E2 1092.101} C_VEL
LIN {X 0,Y 323.506,Z 1045.839,A -85,B 0,C 180,E1 1090.626,E2 1090.626} C_VEL
LIN {X 0,Y 341.197,Z 1023.017,A -85,B 0,C 180,E1 1089.043,E2 1089.043} C_VEL
LIN {X 0,Y 353.916,Z 1004.523,A -85,B 0,C 180,E1 1088.02,E2 1088.02} C_VEL
LIN {X 0,Y 364.833,Z 986.951,A -85,B 0,C 180,E1 1087.204,E2 1087.204} C_VEL
LIN {X 0,Y 376.781,Z 965.47,A -85,B 0,C 180,E1 1086.374,E2 1086.374} C_VEL
LIN {X 0,Y 388.805,Z 940.308,A -85,B 0,C 180,E1 1085.599,E2 1085.599} C_VEL
LIN {X 0,Y 397.025,Z 920.347,A -85,B 0,C 180,E1 1085.107,E2 1085.107} C_VEL
LIN {X 0,Y 404.295,Z 899.914,A -85,B 0,C 180,E1 1084.679,E2 1084.679} C_VEL
LIN {X 0,Y 411.494,Z 875.864,A -85,B 0,C 180,E1 1084.289,E2 1084.289} C_VEL
LIN {X 0,Y 417.803,Z 848.345,A -85,B 0,C 180,E1 1083.929,E2 1083.929} C_VEL
LIN {X 0,Y 421.607,Z 825.799,A -85,B 0,C 180,E1 1083.657,E2 1083.657} C_VEL
LIN {X 0,Y 438.81,Z 685.529,A -85,B 0,C 180,E1 1082.031,E2 1082.031} C_VEL
LIN {X 0,Y 438.807,Z 685.637,A -85,B 0,C 180,E1 1081.388,E2 1081.388} C_VEL
LIN {X 0,Y 426.948,Z 783.545,A -85,B 0,C 180,E1 1080.211,E2 1080.211} C_VEL
LIN {X 0,Y 426.019,Z 791.252,A -85,B 0,C 180,E1 1080.255,E2 1080.255} C_VEL
LIN {X 0,Y 423.43,Z 811.87,A -85,B 0,C 180,E1 1080.858,E2 1080.858} C_VEL
LIN {X 0,Y 422.516,Z 818.461,A -85,B 0,C 180,E1 1080.876,E2 1080.876} C_VEL
LIN {X 0,Y 418.467,Z 843.861,A -85,B 0,C 180,E1 1080.569,E2 1080.569} C_VEL
LIN {X 0,Y 413.671,Z 866.149,A -85,B 0,C 180,E1 1080.292,E2 1080.292} C_VEL
LIN {X 0,Y 406.636,Z 891.983,A -85,B 0,C 180,E1 1079.911,E2 1079.911} C_VEL
LIN {X 0,Y 397.968,Z 916.956,A -85,B 0,C 180,E1 1079.437,E2 1079.437} C_VEL
LIN {X 0,Y 389.516,Z 937.724,A -85,B 0,C 180,E1 1078.949,E2 1078.949} C_VEL
LIN {X 0,Y 379.542,Z 959.088,A -85,B 0,C 180,E1 1078.339,E2 1078.339} C_VEL
LIN {X 0,Y 365.817,Z 984.418,A -85,B 0,C 180,E1 1077.444,E2 1077.444} C_VEL
LIN {X 0,Y 353.584,Z 1004.163,A -85,B 0,C 180,E1 1076.579,E2 1076.579} C_VEL
LIN {X 0,Y 340.954,Z 1022.517,A -85,B 0,C 180,E1 1075.614,E2 1075.614} C_VEL
LIN {X 0,Y 324.603,Z 1043.913,A -85,B 0,C 180,E1 1074.229,E2 1074.229} C_VEL
LIN {X 0,Y 307.984,Z 1063.11,A -85,B 0,C 180,E1 1072.66,E2 1072.66} C_VEL
LIN {X 0,Y 293.473,Z 1078.419,A -85,B 0,C 180,E1 1071.128,E2 1071.128} C_VEL
LIN {X 0,Y 276.923,Z 1094.452,A -85,B 0,C 180,E1 1069.141,E2 1069.141} C_VEL
LIN {X 0,Y 256.276,Z 1112.508,A -85,B 0,C 180,E1 1066.231,E2 1066.231} C_VEL
LIN {X 0,Y 239.868,Z 1125.559,A -85,B 0,C 180,E1 1063.482,E2 1063.482} C_VEL
LIN {X 0,Y 224.038,Z 1137.262,A -85,B 0,C 180,E1 1060.335,E2 1060.335} C_VEL
LIN {X 0,Y 205.13,Z 1150.309,A -85,B 0,C 180,E1 1055.712,E2 1055.712} C_VEL
LIN {X 0,Y 187.707,Z 1161.282,A -85,B 0,C 180,E1 1050.256,E2 1050.256} C_VEL
LIN {X 0,Y 174.001,Z 1169.553,A -85,B 0,C 180,E1 1044.684,E2 1044.684} C_VEL
LIN {X 0,Y 161.011,Z 1177.232,A -85,B 0,C 180,E1 1037.644,E2 1037.644} C_VEL
LIN {X 0,Y 148.597,Z 1184.613,A -85,B 0,C 180,E1 1027.756,E2 1027.756} C_VEL
LIN {X 0,Y 141.754,Z 1189.045,A -85,B 0,C 180,E1 1018.995,E2 1018.995} C_VEL
LIN {X 0,Y 137.896,Z 1192.073,A -85,B 0,C 180,E1 1010.367,E2 1010.367} C_VEL
LIN {X 0,Y 136.3,Z 1193.918,A -85,B 0,C 180,E1 1002.282,E2 1002.282} C_VEL
LIN {X 0,Y 136.03,Z 1194.787,A -85,B 0,C 180,E1 995.482,E2 995.482} C_VEL
LIN {X 0,Y 136.051,Z 1195.054,A -85,B 0,C 180,E1 989.157,E2 989.157} C_VEL
LIN {X 0,Y 136.065,Z 1194.623,A -85,B 0,C 180,E1 981.973,E2 981.973} C_VEL
LIN {X 0,Y 137.208,Z 1192.779,A -85,B 0,C 180,E1 972.177,E2 972.177} C_VEL
LIN {X 0,Y 140.874,Z 1189.641,A -85,B 0,C 180,E1 962.525,E2 962.525} C_VEL
LIN {X 0,Y 146.809,Z 1185.656,A -85,B 0,C 180,E1 954.144,E2 954.144} C_VEL
LIN {X 0,Y 155.193,Z 1180.56,A -85,B 0,C 180,E1 946.418,E2 946.418} C_VEL
LIN {X 0,Y 167.501,Z 1173.376,A -85,B 0,C 180,E1 938.556,E2 938.556} C_VEL
LIN {X 0,Y 183.625,Z 1163.7,A -85,B 0,C 180,E1 931.25,E2 931.25} C_VEL
LIN {X 0,Y 198.392,Z 1154.458,A -85,B 0,C 180,E1 926.219,E2 926.219} C_VEL
LIN {X 0,Y 213.624,Z 1144.397,A -85,B 0,C 180,E1 922.065,E2 922.065} C_VEL
LIN {X 0,Y 233.129,Z 1130.604,A -85,B 0,C 180,E1 917.795,E2 917.795} C_VEL
LIN {X 0,Y 251.655,Z 1116.102,A -85,B 0,C 180,E1 914.496,E2 914.496} C_VEL
LIN {X 0,Y 266.988,Z 1103.145,A -85,B 0,C 180,E1 912.188,E2 912.188} C_VEL
LIN {X 0,Y 283.316,Z 1088.201,A -85,B 0,C 180,E1 910.052,E2 910.052} C_VEL
LIN {X 0,Y 303.275,Z 1067.978,A -85,B 0,C 180,E1 907.806,E2 907.806} C_VEL
LIN {X 0,Y 318.45,Z 1050.857,A -85,B 0,C 180,E1 906.309,E2 906.309} C_VEL
LIN {X 0,Y 332.27,Z 1033.768,A -85,B 0,C 180,E1 905.088,E2 905.088} C_VEL
LIN {X 0,Y 347.746,Z 1012.649,A -85,B 0,C 180,E1 903.854,E2 903.854} C_VEL
LIN {X 0,Y 361.893,Z 990.51,A -85,B 0,C 180,E1 902.813,E2 902.813} C_VEL
LIN {X 0,Y 372.856,Z 971.326,A -85,B 0,C 180,E1 902.073,E2 902.073} C_VEL
LIN {X 0,Y 383.074,Z 951.244,A -85,B 0,C 180,E1 901.428,E2 901.428} C_VEL
LIN {X 0,Y 394.488,Z 925.272,A -85,B 0,C 180,E1 900.752,E2 900.752} C_VEL
LIN {X 0,Y 402.957,Z 902.133,A -85,B 0,C 180,E1 900.271,E2 900.271} C_VEL
LIN {X 0,Y 409.577,Z 880.665,A -85,B 0,C 180,E1 899.912,E2 899.912} C_VEL
LIN {X 0,Y 416.182,Z 854.257,A -85,B 0,C 180,E1 899.56,E2 899.56} C_VEL
LIN {X 0,Y 420.878,Z 827.721,A -85,B 0,C 180,E1 899.236,E2 899.236} C_VEL
LIN {X 0,Y 431.169,Z 745.271,A -85,B 0,C 180,E1 898.257,E2 898.257} C_VEL
LIN {X 0,Y 420.543,Z 829.806,A -85,B 0,C 180,E1 897.297,E2 897.297} C_VEL
LIN {X 0,Y 415.179,Z 858.425,A -85,B 0,C 180,E1 896.96,E2 896.96} C_VEL
LIN {X 0,Y 409.245,Z 881.72,A -85,B 0,C 180,E1 896.652,E2 896.652} C_VEL
LIN {X 0,Y 402.528,Z 903.315,A -85,B 0,C 180,E1 896.309,E2 896.309} C_VEL
LIN {X 0,Y 393.02,Z 928.884,A -85,B 0,C 180,E1 895.778,E2 895.778} C_VEL
LIN {X 0,Y 382.323,Z 952.642,A -85,B 0,C 180,E1 895.152,E2 895.152} C_VEL
LIN {X 0,Y 372.639,Z 971.533,A -85,B 0,C 180,E1 894.553,E2 894.553} C_VEL
LIN {X 0,Y 361.081,Z 991.606,A -85,B 0,C 180,E1 893.784,E2 893.784} C_VEL
LIN {X 0,Y 345.308,Z 1015.626,A -85,B 0,C 180,E1 892.636,E2 892.636} C_VEL
LIN {X 0,Y 332.047,Z 1033.498,A -85,B 0,C 180,E1 891.572,E2 891.572} C_VEL
LIN {X 0,Y 318.44,Z 1050.149,A -85,B 0,C 180,E1 890.381,E2 890.381} C_VEL
LIN {X 0,Y 301.48,Z 1068.996,A -85,B 0,C 180,E1 888.715,E2 888.715} C_VEL
LIN {X 0,Y 283.563,Z 1086.656,A -85,B 0,C 180,E1 886.709,E2 886.709} C_VEL
LIN {X 0,Y 267.529,Z 1101.046,A -85,B 0,C 180,E1 884.638,E2 884.638} C_VEL
LIN {X 0,Y 250.679,Z 1114.917,A -85,B 0,C 180,E1 882.113,E2 882.113} C_VEL
LIN {X 0,Y 230.126,Z 1130.19,A -85,B 0,C 180,E1 878.407,E2 878.407} C_VEL
LIN {X 0,Y 213.937,Z 1141.136,A -85,B 0,C 180,E1 874.829,E2 874.829} C_VEL
LIN {X 0,Y 198.47,Z 1150.863,A -85,B 0,C 180,E1 870.641,E2 870.641} C_VEL
LIN {X 0,Y 180.675,Z 1161.268,A -85,B 0,C 180,E1 864.442,E2 864.442} C_VEL
LIN {X 0,Y 166.879,Z 1168.773,A -85,B 0,C 180,E1 857.986,E2 857.986} C_VEL
LIN {X 0,Y 156.221,Z 1174.434,A -85,B 0,C 180,E1 851.243,E2 851.243} C_VEL
LIN {X 0,Y 146.708,Z 1179.572,A -85,B 0,C 180,E1 842.577,E2 842.577} C_VEL
LIN {X 0,Y 139.73,Z 1183.588,A -85,B 0,C 180,E1 831.846,E2 831.846} C_VEL
LIN {X 0,Y 137.003,Z 1185.527,A -85,B 0,C 180,E1 823.077,E2 823.077} C_VEL
LIN {X 0,Y 136.172,Z 1186.413,A -85,B 0,C 180,E1 815.478,E2 815.478} C_VEL
LIN {X 0,Y 136.092,Z 1186.611,A -85,B 0,C 180,E1 808.317,E2 808.317} C_VEL
LIN {X 0,Y 136.493,Z 1186.063,A -85,B 0,C 180,E1 800.301,E2 800.301} C_VEL
LIN {X 0,Y 138.544,Z 1184.385,A -85,B 0,C 180,E1 791.05,E2 791.05} C_VEL
LIN {X 0,Y 142.791,Z 1181.755,A -85,B 0,C 180,E1 782.475,E2 782.475} C_VEL
LIN {X 0,Y 149.847,Z 1177.88,A -85,B 0,C 180,E1 774.043,E2 774.043} C_VEL
LIN {X 0,Y 161.468,Z 1171.83,A -85,B 0,C 180,E1 765.096,E2 765.096} C_VEL
LIN {X 0,Y 175.55,Z 1164.158,A -85,B 0,C 180,E1 757.656,E2 757.656} C_VEL
LIN {X 0,Y 189.301,Z 1156.394,A -85,B 0,C 180,E1 752.241,E2 752.241} C_VEL
LIN {X 0,Y 206.483,Z 1146.115,A -85,B 0,C 180,E1 747.001,E2 747.001} C_VEL
LIN {X 0,Y 225.169,Z 1133.78,A -85,B 0,C 180,E1 742.538,E2 742.538} C_VEL
LIN {X 0,Y 240.774,Z 1122.617,A -85,B 0,C 180,E1 739.495,E2 739.495} C_VEL
LIN {X 0,Y 256.963,Z 1110.076,A -85,B 0,C 180,E1 736.822,E2 736.822} C_VEL
LIN {X 0,Y 276.314,Z 1093.629,A -85,B 0,C 180,E1 734.121,E2 734.121} C_VEL
LIN {X 0,Y 293.452,Z 1077.328,A -85,B 0,C 180,E1 732.072,E2 732.072} C_VEL
LIN {X 0,Y 308.144,Z 1062.043,A -85,B 0,C 180,E1 730.524,E2 730.524} C_VEL
LIN {X 0,Y 323.983,Z 1043.964,A -85,B 0,C 180,E1 729.041,E2 729.041} C_VEL
LIN {X 0,Y 340.493,Z 1022.712,A -85,B 0,C 180,E1 727.658,E2 727.658} C_VEL
LIN {X 0,Y 353.359,Z 1004.176,A -85,B 0,C 180,E1 726.688,E2 726.688} C_VEL
LIN {X 0,Y 364.875,Z 985.752,A -85,B 0,C 180,E1 725.883,E2 725.883} C_VEL
LIN {X 0,Y 377.912,Z 962.286,A -85,B 0,C 180,E1 725.04,E2 725.04} C_VEL
LIN {X 0,Y 389.078,Z 938.614,A -85,B 0,C 180,E1 724.365,E2 724.365} C_VEL
LIN {X 0,Y 397.531,Z 917.998,A -85,B 0,C 180,E1 723.894,E2 723.894} C_VEL
LIN {X 0,Y 405.381,Z 895.662,A -85,B 0,C 180,E1 723.469,E2 723.469} C_VEL
LIN {X 0,Y 413.256,Z 867.771,A -85,B 0,C 180,E1 723.063,E2 723.063} C_VEL
LIN {X 0,Y 418.223,Z 844.976,A -85,B 0,C 180,E1 722.789,E2 722.789} C_VEL
LIN {X 0,Y 422.04,Z 821.551,A -85,B 0,C 180,E1 722.517,E2 722.517} C_VEL
LIN {X 0,Y 430.995,Z 749.198,A -85,B 0,C 180,E1 721.694,E2 721.694} C_VEL
LIN {X 0,Y 422.516,Z 818.461,A -85,B 0,C 180,E1 720.876,E2 720.876} C_VEL
LIN {X 0,Y 421.332,Z 826.624,A -85,B 0,C 180,E1 720.908,E2 720.908} C_VEL
LIN {X 0,Y 417.65,Z 848.449,A -85,B 0,C 180,E1 721.508,E2 721.508} C_VEL
LIN {X 0,Y 416.126,Z 855.36,A -85,B 0,C 180,E1 721.533,E2 721.533} C_VEL
LIN {X 0,Y 409.601,Z 881.082,A -85,B 0,C 180,E1 721.207,E2 721.207} C_VEL
LIN {X 0,Y 402.995,Z 902.307,A -85,B 0,C 180,E1 720.873,E2 720.873} C_VEL
LIN {X 0,Y 394.46,Z 925.415,A -85,B 0,C 180,E1 720.42,E2 720.42} C_VEL
LIN {X 0,Y 382.953,Z 951.337,A -85,B 0,C 180,E1 719.783,E2 719.783} C_VEL
LIN {X 0,Y 372.491,Z 971.685,A -85,B 0,C 180,E1 719.166,E2 719.166} C_VEL
LIN {X 0,Y 361.086,Z 991.394,A -85,B 0,C 180,E1 718.444,E2 718.444} C_VEL
LIN {X 0,Y 345.814,Z 1014.714,A -85,B 0,C 180,E1 717.39,E2 717.39} C_VEL
LIN {X 0,Y 331.151,Z 1034.387,A -85,B 0,C 180,E1 716.29,E2 716.29} C_VEL
LIN {X 0,Y 317.001,Z 1051.59,A -85,B 0,C 180,E1 715.115,E2 715.115} C_VEL
LIN {X 0,Y 299.546,Z 1070.872,A -85,B 0,C 180,E1 713.483,E2 713.483} C_VEL
LIN {X 0,Y 281.044,Z 1088.997,A -85,B 0,C 180,E1 711.509,E2 711.509} C_VEL
LIN {X 0,Y 265.344,Z 1103.064,A -85,B 0,C 180,E1 709.577,E2 709.577} C_VEL
LIN {X 0,Y 248.764,Z 1116.738,A -85,B 0,C 180,E1 707.228,E2 707.228} C_VEL
LIN {X 0,Y 228.035,Z 1132.349,A -85,B 0,C 180,E1 703.702,E2 703.702} C_VEL
LIN {X 0,Y 209.785,Z 1144.774,A -85,B 0,C 180,E1 699.873,E2 699.873} C_VEL
LIN {X 0,Y 194.042,Z 1154.769,A -85,B 0,C 180,E1 695.79,E2 695.79} C_VEL
LIN {X 0,Y 175.929,Z 1165.617,A -85,B 0,C 180,E1 689.753,E2 689.753} C_VEL
LIN {X 0,Y 159.996,Z 1174.446,A -85,B 0,C 180,E1 682.529,E2 682.529} C_VEL
LIN {X 0,Y 148.734,Z 1180.622,A -85,B 0,C 180,E1 675.445,E2 675.445} C_VEL
LIN {X 0,Y 139.697,Z 1185.694,A -85,B 0,C 180,E1 667.392,E2 667.392} C_VEL
LIN {X 0,Y 132.855,Z 1189.928,A -85,B 0,C 180,E1 657.814,E2 657.814} C_VEL
LIN {X 0,Y 128.919,Z 1193.069,A -85,B 0,C 180,E1 646.675,E2 646.675} C_VEL
LIN {X 0,Y 128.047,Z 1194.46,A -85,B 0,C 180,E1 637.176,E2 637.176} C_VEL
LIN {X 0,Y 128.06,Z 1194.849,A -85,B 0,C 180,E1 629.999,E2 629.999} C_VEL
LIN {X 0,Y 128.052,Z 1194.442,A -85,B 0,C 180,E1 622.603,E2 622.603} C_VEL
LIN {X 0,Y 129.014,Z 1192.979,A -85,B 0,C 180,E1 612.871,E2 612.871} C_VEL
LIN {X 0,Y 133.091,Z 1189.723,A -85,B 0,C 180,E1 601.75,E2 601.75} C_VEL
LIN {X 0,Y 139.755,Z 1185.615,A -85,B 0,C 180,E1 592.544,E2 592.544} C_VEL
LIN {X 0,Y 148.734,Z 1180.565,A -85,B 0,C 180,E1 584.553,E2 584.553} C_VEL
LIN {X 0,Y 160.584,Z 1174.06,A -85,B 0,C 180,E1 577.155,E2 577.155} C_VEL
LIN {X 0,Y 178.683,Z 1163.849,A -85,B 0,C 180,E1 569.196,E2 569.196} C_VEL
LIN {X 0,Y 194.804,Z 1154.188,A -85,B 0,C 180,E1 563.987,E2 563.987} C_VEL
LIN {X 0,Y 210.596,Z 1144.126,A -85,B 0,C 180,E1 559.934,E2 559.934} C_VEL
LIN {X 0,Y 230.687,Z 1130.322,A -85,B 0,C 180,E1 555.797,E2 555.797} C_VEL
LIN {X 0,Y 249.08,Z 1116.295,A -85,B 0,C 180,E1 552.714,E2 552.714} C_VEL
LIN {X 0,Y 264.427,Z 1103.637,A -85,B 0,C 180,E1 550.535,E2 550.535} C_VEL
LIN {X 0,Y 280.109,Z 1089.622,A -85,B 0,C 180,E1 548.588,E2 548.588} C_VEL
LIN {X 0,Y 298.928,Z 1071.256,A -85,B 0,C 180,E1 546.569,E2 546.569} C_VEL
LIN {X 0,Y 316.142,Z 1052.277,A -85,B 0,C 180,E1 544.95,E2 544.95} C_VEL
LIN {X 0,Y 330.178,Z 1035.266,A -85,B 0,C 180,E1 543.777,E2 543.777} C_VEL
LIN {X 0,Y 343.362,Z 1017.698,A -85,B 0,C 180,E1 542.773,E2 542.773} C_VEL
LIN {X 0,Y 358.806,Z 994.696,A -85,B 0,C 180,E1 541.696,E2 541.696} C_VEL
LIN {X 0,Y 371.5,Z 972.966,A -85,B 0,C 180,E1 540.883,E2 540.883} C_VEL
LIN {X 0,Y 381.459,Z 953.783,A -85,B 0,C 180,E1 540.29,E2 540.29} C_VEL
LIN {X 0,Y 390.957,Z 933.054,A -85,B 0,C 180,E1 539.756,E2 539.756} C_VEL
LIN {X 0,Y 401.492,Z 905.877,A -85,B 0,C 180,E1 539.194,E2 539.194} C_VEL
LIN {X 0,Y 408.701,Z 883.162,A -85,B 0,C 180,E1 538.823,E2 538.823} C_VEL
LIN {X 0,Y 414.461,Z 861.047,A -85,B 0,C 180,E1 538.535,E2 538.535} C_VEL
LIN {X 0,Y 418.858,Z 839.746,A -85,B 0,C 180,E1 538.279,E2 538.279} C_VEL
LIN {X 0,Y 413.888,Z 863.418,A -85,B 0,C 180,E1 538.01,E2 538.01} C_VEL
LIN {X 0,Y 408.147,Z 885.055,A -85,B 0,C 180,E1 537.73,E2 537.73} C_VEL
LIN {X 0,Y 399.809,Z 910.748,A -85,B 0,C 180,E1 537.32,E2 537.32} C_VEL
LIN {X 0,Y 389.932,Z 935.327,A -85,B 0,C 180,E1 536.809,E2 536.809} C_VEL
LIN {X 0,Y 380.751,Z 955.134,A -85,B 0,C 180,E1 536.295,E2 536.295} C_VEL
LIN {X 0,Y 370.502,Z 974.662,A -85,B 0,C 180,E1 535.694,E2 535.694} C_VEL
LIN {X 0,Y 355.456,Z 999.677,A -85,B 0,C 180,E1 534.738,E2 534.738} C_VEL
LIN {X 0,Y 342.442,Z 1018.633,A -85,B 0,C 180,E1 533.832,E2 533.832} C_VEL
LIN {X 0,Y 329.527,Z 1035.646,A -85,B 0,C 180,E1 532.846,E2 532.846} C_VEL
LIN {X 0,Y 314.354,Z 1053.765,A -85,B 0,C 180,E1 531.577,E2 531.577} C_VEL
LIN {X 0,Y 295.632,Z 1073.641,A -85,B 0,C 180,E1 529.807,E2 529.807} C_VEL
LIN {X 0,Y 279.966,Z 1088.614,A -85,B 0,C 180,E1 528.119,E2 528.119} C_VEL
LIN {X 0,Y 263.682,Z 1102.848,A -85,B 0,C 180,E1 526.109,E2 526.109} C_VEL
LIN {X 0,Y 243.413,Z 1118.909,A -85,B 0,C 180,E1 523.159,E2 523.159} C_VEL
LIN {X 0,Y 225.549,Z 1131.584,A -85,B 0,C 180,E1 520.022,E2 520.022} C_VEL
LIN {X 0,Y 209.879,Z 1141.831,A -85,B 0,C 180,E1 516.708,E2 516.708} C_VEL
LIN {X 0,Y 193.056,Z 1152.023,A -85,B 0,C 180,E1 512.332,E2 512.332} C_VEL
LIN {X 0,Y 174.651,Z 1162.211,A -85,B 0,C 180,E1 506.113,E2 506.113} C_VEL
LIN {X 0,Y 160.879,Z 1169.323,A -85,B 0,C 180,E1 499.86,E2 499.86} C_VEL
LIN {X 0,Y 149.63,Z 1174.934,A -85,B 0,C 180,E1 492.97,E2 492.97} C_VEL
LIN {X 0,Y 138.797,Z 1180.417,A -85,B 0,C 180,E1 483.196,E2 483.196} C_VEL
LIN {X 0,Y 131.8,Z 1184.053,A -85,B 0,C 180,E1 472.292,E2 472.292} C_VEL
LIN {X 0,Y 129.051,Z 1185.84,A -85,B 0,C 180,E1 463.442,E2 463.442} C_VEL
LIN {X 0,Y 128.17,Z 1186.681,A -85,B 0,C 180,E1 455.373,E2 455.373} C_VEL
LIN {X 0,Y 128.096,Z 1186.858,A -85,B 0,C 180,E1 448.212,E2 448.212} C_VEL
LIN {X 0,Y 128.561,Z 1186.312,A -85,B 0,C 180,E1 439.696,E2 439.696} C_VEL
LIN {X 0,Y 130.879,Z 1184.636,A -85,B 0,C 180,E1 429.893,E2 429.893} C_VEL
LIN {X 0,Y 135.582,Z 1182.009,A -85,B 0,C 180,E1 420.875,E2 420.875} C_VEL
LIN {X 0,Y 142.857,Z 1178.333,A -85,B 0,C 180,E1 412.489,E2 412.489} C_VEL
LIN {X 0,Y 154.649,Z 1172.592,A -85,B 0,C 180,E1 403.604,E2 403.604} C_VEL
LIN {X 0,Y 169.978,Z 1164.758,A -85,B 0,C 180,E1 395.732,E2 395.732} C_VEL
LIN {X 0,Y 184.359,Z 1157.016,A -85,B 0,C 180,E1 390.291,E2 390.291} C_VEL
LIN {X 0,Y 200.536,Z 1147.719,A -85,B 0,C 180,E1 385.517,E2 385.517} C_VEL
LIN {X 0,Y 221.311,Z 1134.606,A -85,B 0,C 180,E1 380.738,E2 380.738} C_VEL
LIN {X 0,Y 238.151,Z 1122.884,A -85,B 0,C 180,E1 377.626,E2 377.626} C_VEL
LIN {X 0,Y 254.706,Z 1110.348,A -85,B 0,C 180,E1 375.052,E2 375.052} C_VEL
LIN {X 0,Y 274.43,Z 1093.917,A -85,B 0,C 180,E1 372.461,E2 372.461} C_VEL
LIN {X 0,Y 291.853,Z 1077.624,A -85,B 0,C 180,E1 370.504,E2 370.504} C_VEL
LIN {X 0,Y 306.292,Z 1062.849,A -85,B 0,C 180,E1 369.073,E2 369.073} C_VEL
LIN {X 0,Y 321.382,Z 1045.927,A -85,B 0,C 180,E1 367.735,E2 367.735} C_VEL
LIN {X 0,Y 339.509,Z 1023.069,A -85,B 0,C 180,E1 366.305,E2 366.305} C_VEL
LIN {X 0,Y 352.765,Z 1004.171,A -85,B 0,C 180,E1 365.367,E2 365.367} C_VEL
LIN {X 0,Y 364.138,Z 986.16,A -85,B 0,C 180,E1 364.624,E2 364.624} C_VEL
LIN {X 0,Y 377.293,Z 962.767,A -85,B 0,C 180,E1 363.828,E2 363.828} C_VEL
LIN {X 0,Y 388.551,Z 939.158,A -85,B 0,C 180,E1 363.189,E2 363.189} C_VEL
LIN {X 0,Y 397.123,Z 918.475,A -85,B 0,C 180,E1 362.742,E2 362.742} C_VEL
LIN {X 0,Y 404.549,Z 897.645,A -85,B 0,C 180,E1 362.363,E2 362.363} C_VEL
LIN {X 0,Y 412.66,Z 869.815,A -85,B 0,C 180,E1 361.974,E2 361.974} C_VEL
LIN {X 0,Y 417.979,Z 845.912,A -85,B 0,C 180,E1 361.7,E2 361.7} C_VEL
LIN {X 0,Y 418.373,Z 843.862,A -85,B 0,C 180,E1 361.668,E2 361.668} C_VEL
LIN {X 0,Y 416.126,Z 855.36,A -85,B 0,C 180,E1 361.533,E2 361.533} C_VEL
LIN {X 0,Y 416.068,Z 855.851,A -85,B 0,C 180,E1 361.53,E2 361.53} C_VEL
LIN {X 0,Y 416.068,Z 939.678,A -85,B 0,C 180,E1 361.53,E2 361.53} C_VEL
LIN {X 0,Y 401.113,Z 939.678,A -85,B 0,C 180,E1 361.798,E2 361.798} C_VEL
LIN {X 0,Y 399.13,Z 937.678,A -85,B 0,C 180,E1 361.835,E2 361.835} C_VEL
LIN {X 0,Y 399.13,Z 923.251,A -85,B 0,C 180,E1 361.835,E2 361.835} C_VEL
LIN {X 0,Y 395.499,Z 922.488,A -85,B 0,C 180,E1 361.651,E2 361.651} C_VEL
LIN {X 0,Y 384.016,Z 948.806,A -85,B 0,C 180,E1 361.059,E2 361.059} C_VEL
LIN {X 0,Y 372.963,Z 970.32,A -85,B 0,C 180,E1 360.455,E2 360.455} C_VEL
LIN {X 0,Y 361.955,Z 989.334,A -85,B 0,C 180,E1 359.811,E2 359.811} C_VEL
LIN {X 0,Y 348.512,Z 1010.084,A -85,B 0,C 180,E1 358.957,E2 358.957} C_VEL
LIN {X 0,Y 332.195,Z 1032.195,A -85,B 0,C 180,E1 357.832,E2 357.832} C_VEL
LIN {X 0,Y 317.485,Z 1050.013,A -85,B 0,C 180,E1 356.7,E2 356.7} C_VEL
LIN {X 0,Y 302.913,Z 1066.08,A -85,B 0,C 180,E1 355.454,E2 355.454} C_VEL
LIN {X 0,Y 284.684,Z 1084.39,A -85,B 0,C 180,E1 353.697,E2 353.697} C_VEL
LIN {X 0,Y 265.427,Z 1101.535,A -85,B 0,C 180,E1 351.552,E2 351.552} C_VEL
LIN {X 0,Y 249.185,Z 1114.77,A -85,B 0,C 180,E1 349.444,E2 349.444} C_VEL
LIN {X 0,Y 231.179,Z 1128.255,A -85,B 0,C 180,E1 346.691,E2 346.691} C_VEL
LIN {X 0,Y 209.551,Z 1142.921,A -85,B 0,C 180,E1 342.61,E2 342.61} C_VEL
LIN {X 0,Y 192.319,Z 1153.557,A -85,B 0,C 180,E1 338.531,E2 338.531} C_VEL
LIN {X 0,Y 176.187,Z 1162.845,A -85,B 0,C 180,E1 333.721,E2 333.721} C_VEL
LIN {X 0,Y 158.185,Z 1172.608,A -85,B 0,C 180,E1 326.548,E2 326.548} C_VEL
LIN {X 0,Y 144.017,Z 1179.83,A -85,B 0,C 180,E1 318.573,E2 318.573} C_VEL
LIN {X 0,Y 134.037,Z 1184.971,A -85,B 0,C 180,E1 310.456,E2 310.456} C_VEL
LIN {X 0,Y 126.685,Z 1188.995,A -85,B 0,C 180,E1 301.392,E2 301.392} C_VEL
LIN {X 0,Y 121.987,Z 1192.054,A -85,B 0,C 180,E1 291.139,E2 291.139} C_VEL
LIN {X 0,Y 120.136,Z 1194.007,A -85,B 0,C 180,E1 280.065,E2 280.065} C_VEL
LIN {X 0,Y 120.046,Z 1194.493,A -85,B 0,C 180,E1 272.386,E2 272.386} C_VEL
LIN {X 0,Y 120.035,Z 1194.414,A -85,B 0,C 180,E1 266.178,E2 266.178} C_VEL
LIN {X 0,Y 120.226,Z 1193.771,A -85,B 0,C 180,E1 258.485,E2 258.485} C_VEL
LIN {X 0,Y 122.133,Z 1191.906,A -85,B 0,C 180,E1 248.382,E2 248.382} C_VEL
LIN {X 0,Y 126.838,Z 1188.867,A -85,B 0,C 180,E1 238.363,E2 238.363} C_VEL
LIN {X 0,Y 134.042,Z 1184.921,A -85,B 0,C 180,E1 229.535,E2 229.535} C_VEL
LIN {X 0,Y 144.551,Z 1179.505,A -85,B 0,C 180,E1 221.064,E2 221.064} C_VEL
LIN {X 0,Y 160.783,Z 1171.136,A -85,B 0,C 180,E1 212.246,E2 212.246} C_VEL
LIN {X 0,Y 176.926,Z 1162.327,A -85,B 0,C 180,E1 206.028,E2 206.028} C_VEL
LIN {X 0,Y 192.318,Z 1153.447,A -85,B 0,C 180,E1 201.464,E2 201.464} C_VEL
LIN {X 0,Y 209.549,Z 1142.795,A -85,B 0,C 180,E1 197.384,E2 197.384} C_VEL
LIN {X 0,Y 231.627,Z 1127.758,A -85,B 0,C 180,E1 193.226,E2 193.226} C_VEL
LIN {X 0,Y 248.281,Z 1115.283,A -85,B 0,C 180,E1 190.676,E2 190.676} C_VEL
LIN {X 0,Y 264.882,Z 1101.775,A -85,B 0,C 180,E1 188.505,E2 188.505} C_VEL
LIN {X 0,Y 283.731,Z 1085.025,A -85,B 0,C 180,E1 186.392,E2 186.392} C_VEL
LIN {X 0,Y 301.947,Z 1066.82,A -85,B 0,C 180,E1 184.623,E2 184.623} C_VEL
LIN {X 0,Y 316.997,Z 1050.253,A -85,B 0,C 180,E1 183.328,E2 183.328} C_VEL
LIN {X 0,Y 331.212,Z 1033.064,A -85,B 0,C 180,E1 182.229,E2 182.229} C_VEL
LIN {X 0,Y 347.664,Z 1010.909,A -85,B 0,C 180,E1 181.088,E2 181.088} C_VEL
LIN {X 0,Y 361.46,Z 989.654,A -85,B 0,C 180,E1 180.207,E2 180.207} C_VEL
LIN {X 0,Y 372.968,Z 969.769,A -85,B 0,C 180,E1 179.532,E2 179.532} C_VEL
LIN {X 0,Y 385.028,Z 946.154,A -85,B 0,C 180,E1 178.877,E2 178.877} C_VEL
LIN {X 0,Y 395.571,Z 921.515,A -85,B 0,C 180,E1 178.332,E2 178.332} C_VEL
LIN {X 0,Y 396.127,Z 920.083,A -85,B 0,C 180,E1 178.3,E2 178.3} C_VEL
LIN {X 0,Y 386.583,Z 942.653,A -85,B 0,C 180,E1 177.828,E2 177.828} C_VEL
LIN {X 0,Y 373.816,Z 968.17,A -85,B 0,C 180,E1 177.151,E2 177.151} C_VEL
LIN {X 0,Y 362.631,Z 987.625,A -85,B 0,C 180,E1 176.507,E2 176.507} C_VEL
LIN {X 0,Y 350.907,Z 1005.882,A -85,B 0,C 180,E1 175.786,E2 175.786} C_VEL
LIN {X 0,Y 335.374,Z 1027.561,A -85,B 0,C 180,E1 174.739,E2 174.739} C_VEL
LIN {X 0,Y 319.003,Z 1047.509,A -85,B 0,C 180,E1 173.517,E2 173.517} C_VEL
LIN {X 0,Y 304.697,Z 1063.306,A -85,B 0,C 180,E1 172.322,E2 172.322} C_VEL
LIN {X 0,Y 289.6,Z 1078.512,A -85,B 0,C 180,E1 170.915,E2 170.915} C_VEL
LIN {X 0,Y 270.085,Z 1096.3,A -85,B 0,C 180,E1 168.831,E2 168.831} C_VEL
LIN {X 0,Y 251.873,Z 1111.06,A -85,B 0,C 180,E1 166.557,E2 166.557} C_VEL
LIN {X 0,Y 234.993,Z 1123.549,A -85,B 0,C 180,E1 164.075,E2 164.075} C_VEL
LIN {X 0,Y 216.081,Z 1136.35,A -85,B 0,C 180,E1 160.732,E2 160.732} C_VEL
LIN {X 0,Y 196.412,Z 1148.256,A -85,B 0,C 180,E1 156.396,E2 156.396} C_VEL
LIN {X 0,Y 180.209,Z 1157.228,A -85,B 0,C 180,E1 151.86,E2 151.86} C_VEL
LIN {X 0,Y 165.373,Z 1164.871,A -85,B 0,C 180,E1 146.552,E2 146.552} C_VEL
LIN {X 0,Y 149.156,Z 1172.744,A -85,B 0,C 180,E1 138.661,E2 138.661} C_VEL
LIN {X 0,Y 136.49,Z 1178.499,A -85,B 0,C 180,E1 129.594,E2 129.594} C_VEL
LIN {X 0,Y 128.541,Z 1182.193,A -85,B 0,C 180,E1 120.891,E2 120.891} C_VEL
LIN {X 0,Y 123.3,Z 1184.839,A -85,B 0,C 180,E1 111.404,E2 111.404} C_VEL
LIN {X 0,Y 120.66,Z 1186.532,A -85,B 0,C 180,E1 100.989,E2 100.989} C_VEL
LIN {X 0,Y 120.096,Z 1187.095,A -85,B 0,C 180,E1 91.909,E2 91.909} C_VEL
LIN {X 0,Y 120.182,Z 1186.938,A -85,B 0,C 180,E1 84.271,E2 84.271} C_VEL
LIN {X 0,Y 121.089,Z 1186.182,A -85,B 0,C 180,E1 76.146,E2 76.146} C_VEL
LIN {X 0,Y 124.049,Z 1184.461,A -85,B 0,C 180,E1 66.738,E2 66.738} C_VEL
LIN {X 0,Y 130.239,Z 1181.456,A -85,B 0,C 180,E1 56.807,E2 56.807} C_VEL
LIN {X 0,Y 142.594,Z 1175.786,A -85,B 0,C 180,E1 45.478,E2 45.478} C_VEL
LIN {X 0,Y 154.977,Z 1170,A -85,B 0,C 180,E1 38.085,E2 38.085} C_VEL
LIN {X 0,Y 168.691,Z 1163.299,A -85,B 0,C 180,E1 32.05,E2 32.05} C_VEL
LIN {X 0,Y 187.203,Z 1153.662,A -85,B 0,C 180,E1 25.975,E2 25.975} C_VEL
LIN {X 0,Y 206.009,Z 1142.685,A -85,B 0,C 180,E1 21.271,E2 21.271} C_VEL
LIN {X 0,Y 222.779,Z 1132.059,A -85,B 0,C 180,E1 17.919,E2 17.919} C_VEL
LIN {X 0,Y 241.964,Z 1118.786,A -85,B 0,C 180,E1 14.77,E2 14.77} C_VEL
LIN {X 0,Y 261.761,Z 1103.408,A -85,B 0,C 180,E1 12.078,E2 12.078} C_VEL
LIN {X 0,Y 278.329,Z 1089.202,A -85,B 0,C 180,E1 10.16,E2 10.16} C_VEL
LIN {X 0,Y 294.236,Z 1074.263,A -85,B 0,C 180,E1 8.555,E2 8.555} C_VEL
LIN {X 0,Y 312.737,Z 1055.026,A -85,B 0,C 180,E1 6.919,E2 6.919} C_VEL
LIN {X 0,Y 328.568,Z 1036.412,A -85,B 0,C 180,E1 5.676,E2 5.676} C_VEL
LIN {X 0,Y 341.627,Z 1019.46,A -85,B 0,C 180,E1 4.746,E2 4.746} C_VEL
LIN {X 0,Y 355.025,Z 1000.195,A -85,B 0,C 180,E1 3.876,E2 3.876} C_VEL
LIN {X 0,Y 369.956,Z 975.719,A -85,B 0,C 180,E1 2.991,E2 2.991} C_VEL
LIN {X 0,Y 380.602,Z 955.669,A -85,B 0,C 180,E1 2.409,E2 2.409} C_VEL
LIN {X 0,Y 390.188,Z 935.175,A -85,B 0,C 180,E1 1.909,E2 1.909} C_VEL
LIN {X 0,Y 395.499,Z 922.488,A -85,B 0,C 180,E1 1.651,E2 1.651} C_VEL
LIN {X 0,Y 399.045,Z 923.267,A -85,B 0,C 180,E1 1.438,E2 1.438} C_VEL
LIN {X 0,Y 399.045,Z 986.654,A -85,B 0,C 180,E1 1.438,E2 1.438} C_VEL
LIN {X 0,Y 377.12,Z 986.654,A -85,B 0,C 180,E1 1.788,E2 1.788} C_VEL
LIN {X 0,Y 375.132,Z 984.654,A -85,B 0,C 180,E1 1.821,E2 1.821} C_VEL
LIN {X 0,Y 375.132,Z 973.597,A -85,B 0,C 180,E1 1.821,E2 1.821} C_VEL
LIN {X 0,Y 371.611,Z 972.584,A -85,B 0,C 180,E1 1.635,E2 1.635} C_VEL
LIN {X 0,Y 359.002,Z 993.844,A -85,B 0,C 180,E1 0.939,E2 0.939} C_VEL
LIN {X 0,Y 343.407,Z 1016.76,A -85,B 0,C 180,E1 0,E2 0} C_VEL
LIN {X 0,Y 329.499,Z 1034.935,A -85,B 0,C 180,E1 -0.91,E2 -0.91} C_VEL
LIN {X 0,Y 315.141,Z 1051.939,A -85,B 0,C 180,E1 -1.95,E2 -1.95} C_VEL
LIN {X 0,Y 296.993,Z 1071.392,A -85,B 0,C 180,E1 -3.428,E2 -3.428} C_VEL
LIN {X 0,Y 278.102,Z 1089.267,A -85,B 0,C 180,E1 -5.187,E2 -5.187} C_VEL
LIN {X 0,Y 261.877,Z 1103.273,A -85,B 0,C 180,E1 -6.926,E2 -6.926} C_VEL
LIN {X 0,Y 244.066,Z 1117.345,A -85,B 0,C 180,E1 -9.138,E2 -9.138} C_VEL
LIN {X 0,Y 221.282,Z 1133.512,A -85,B 0,C 180,E1 -12.578,E2 -12.578} C_VEL
LIN {X 0,Y 203.724,Z 1144.768,A -85,B 0,C 180,E1 -15.855,E2 -15.855} C_VEL
LIN {X 0,Y 186.922,Z 1154.708,A -85,B 0,C 180,E1 -19.705,E2 -19.705} C_VEL
LIN {X 0,Y 167.29,Z 1165.47,A -85,B 0,C 180,E1 -25.511,E2 -25.511} C_VEL
LIN {X 0,Y 149.675,Z 1174.24,A -85,B 0,C 180,E1 -32.679,E2 -32.679} C_VEL
LIN {X 0,Y 136.689,Z 1180.47,A -85,B 0,C 180,E1 -40.07,E2 -40.07} C_VEL
LIN {X 0,Y 125.596,Z 1185.796,A -85,B 0,C 180,E1 -49.248,E2 -49.248} C_VEL
LIN {X 0,Y 116.425,Z 1190.541,A -85,B 0,C 180,E1 -62.202,E2 -62.202} C_VEL
LIN {X 0,Y 112.913,Z 1192.867,A -85,B 0,C 180,E1 -73.016,E2 -73.016} C_VEL
LIN {X 0,Y 112.053,Z 1194.016,A -85,B 0,C 180,E1 -82.825,E2 -82.825} C_VEL
LIN {X 0,Y 112.063,Z 1194.336,A -85,B 0,C 180,E1 -90.512,E2 -90.512} C_VEL
LIN {X 0,Y 112.087,Z 1193.93,A -85,B 0,C 180,E1 -98.724,E2 -98.724} C_VEL
LIN {X 0,Y 113.75,Z 1192.26,A -85,B 0,C 180,E1 -110.587,E2 -110.587} C_VEL
LIN {X 0,Y 119.054,Z 1189.04,A -85,B 0,C 180,E1 -122.515,E2 -122.515} C_VEL
LIN {X 0,Y 127.34,Z 1184.879,A -85,B 0,C 180,E1 -132.477,E2 -132.477} C_VEL
LIN {X 0,Y 138.388,Z 1179.605,A -85,B 0,C 180,E1 -141.053,E2 -141.053} C_VEL
LIN {X 0,Y 154.37,Z 1171.955,A -85,B 0,C 180,E1 -149.482,E2 -149.482} C_VEL
LIN {X 0,Y 172.611,Z 1162.478,A -85,B 0,C 180,E1 -156.241,E2 -156.241} C_VEL
LIN {X 0,Y 189.186,Z 1153.289,A -85,B 0,C 180,E1 -160.872,E2 -160.872} C_VEL
LIN {X 0,Y 207.177,Z 1142.523,A -85,B 0,C 180,E1 -164.85,E2 -164.85} C_VEL
LIN {X 0,Y 229.381,Z 1127.807,A -85,B 0,C 180,E1 -168.751,E2 -168.751} C_VEL
LIN {X 0,Y 246.848,Z 1115.006,A -85,B 0,C 180,E1 -171.245,E2 -171.245} C_VEL
LIN {X 0,Y 263.77,Z 1101.484,A -85,B 0,C 180,E1 -173.301,E2 -173.301} C_VEL
LIN {X 0,Y 283.469,Z 1084.227,A -85,B 0,C 180,E1 -175.347,E2 -175.347} C_VEL
LIN {X 0,Y 301.878,Z 1065.986,A -85,B 0,C 180,E1 -176.998,E2 -176.998} C_VEL
LIN {X 0,Y 316.13,Z 1050.483,A -85,B 0,C 180,E1 -178.135,E2 -178.135} C_VEL
LIN {X 0,Y 330.496,Z 1033.331,A -85,B 0,C 180,E1 -179.171,E2 -179.171} C_VEL
LIN {X 0,Y 346.962,Z 1011.466,A -85,B 0,C 180,E1 -180.232,E2 -180.232} C_VEL
LIN {X 0,Y 361.02,Z 990.047,A -85,B 0,C 180,E1 -181.068,E2 -181.068} C_VEL
LIN {X 0,Y 372.258,Z 970.866,A -85,B 0,C 180,E1 -181.682,E2 -181.682} C_VEL
LIN {X 0,Y 361.243,Z 989.65,A -85,B 0,C 180,E1 -182.277,E2 -182.277} C_VEL
LIN {X 0,Y 346.971,Z 1011.36,A -85,B 0,C 180,E1 -183.112,E2 -183.112} C_VEL
LIN {X 0,Y 330.825,Z 1032.723,A -85,B 0,C 180,E1 -184.14,E2 -184.14} C_VEL
LIN {X 0,Y 316.736,Z 1049.481,A -85,B 0,C 180,E1 -185.138,E2 -185.138} C_VEL
LIN {X 0,Y 301.316,Z 1066.121,A -85,B 0,C 180,E1 -186.354,E2 -186.354} C_VEL
LIN {X 0,Y 280.837,Z 1085.859,A -85,B 0,C 180,E1 -188.198,E2 -188.198} C_VEL
LIN {X 0,Y 263.95,Z 1100.381,A -85,B 0,C 180,E1 -189.963,E2 -189.963} C_VEL
LIN {X 0,Y 247.346,Z 1113.406,A -85,B 0,C 180,E1 -191.965,E2 -191.965} C_VEL
LIN {X 0,Y 227.524,Z 1127.564,A -85,B 0,C 180,E1 -194.801,E2 -194.801} C_VEL
LIN {X 0,Y 206.633,Z 1140.75,A -85,B 0,C 180,E1 -198.48,E2 -198.48} C_VEL
LIN {X 0,Y 189.984,Z 1150.312,A -85,B 0,C 180,E1 -202.136,E2 -202.136} C_VEL
LIN {X 0,Y 172.698,Z 1159.432,A -85,B 0,C 180,E1 -206.921,E2 -206.921} C_VEL
LIN {X 0,Y 153.393,Z 1168.667,A -85,B 0,C 180,E1 -214.122,E2 -214.122} C_VEL
LIN {X 0,Y 139.715,Z 1174.713,A -85,B 0,C 180,E1 -221.284,E2 -221.284} C_VEL
LIN {X 0,Y 128.849,Z 1179.348,A -85,B 0,C 180,E1 -229.318,E2 -229.318} C_VEL
LIN {X 0,Y 119.62,Z 1183.359,A -85,B 0,C 180,E1 -239.898,E2 -239.898} C_VEL
LIN {X 0,Y 113.869,Z 1186.089,A -85,B 0,C 180,E1 -252.628,E2 -252.628} C_VEL
LIN {X 0,Y 112.27,Z 1187.137,A -85,B 0,C 180,E1 -262.836,E2 -262.836} C_VEL
LIN {X 0,Y 112.097,Z 1187.396,A -85,B 0,C 180,E1 -271.021,E2 -271.021} C_VEL
LIN {X 0,Y 112.601,Z 1186.937,A -85,B 0,C 180,E1 -280.746,E2 -280.746} C_VEL
LIN {X 0,Y 115.524,Z 1185.246,A -85,B 0,C 180,E1 -292.384,E2 -292.384} C_VEL
LIN {X 0,Y 121.524,Z 1182.515,A -85,B 0,C 180,E1 -302.889,E2 -302.889} C_VEL
LIN {X 0,Y 130.66,Z 1178.641,A -85,B 0,C 180,E1 -312.33,E2 -312.33} C_VEL
LIN {X 0,Y 144.971,Z 1172.598,A -85,B 0,C 180,E1 -321.837,E2 -321.837} C_VEL
LIN {X 0,Y 161.579,Z 1164.928,A -85,B 0,C 180,E1 -329.332,E2 -329.332} C_VEL
LIN {X 0,Y 177.201,Z 1157.218,A -85,B 0,C 180,E1 -334.529,E2 -334.529} C_VEL
LIN {X 0,Y 194.814,Z 1147.787,A -85,B 0,C 180,E1 -339.083,E2 -339.083} C_VEL
LIN {X 0,Y 216.017,Z 1135.135,A -85,B 0,C 180,E1 -343.361,E2 -343.361} C_VEL
LIN {X 0,Y 233.689,Z 1123.419,A -85,B 0,C 180,E1 -346.227,E2 -346.227} C_VEL
LIN {X 0,Y 250.086,Z 1111.531,A -85,B 0,C 180,E1 -348.468,E2 -348.468} C_VEL
LIN {X 0,Y 269.493,Z 1096.095,A -85,B 0,C 180,E1 -350.719,E2 -350.719} C_VEL
LIN {X 0,Y 288.953,Z 1078.571,A -85,B 0,C 180,E1 -352.644,E2 -352.644} C_VEL
LIN {X 0,Y 304.231,Z 1063.38,A -85,B 0,C 180,E1 -353.963,E2 -353.963} C_VEL
LIN {X 0,Y 319.676,Z 1046.484,A -85,B 0,C 180,E1 -355.155,E2 -355.155} C_VEL
LIN {X 0,Y 338.164,Z 1023.715,A -85,B 0,C 180,E1 -356.424,E2 -356.424} C_VEL
LIN {X 0,Y 351.855,Z 1004.587,A -85,B 0,C 180,E1 -357.266,E2 -357.266} C_VEL
LIN {X 0,Y 363.739,Z 986.092,A -85,B 0,C 180,E1 -357.935,E2 -357.935} C_VEL
LIN {X 0,Y 371.611,Z 972.584,A -85,B 0,C 180,E1 -358.365,E2 -358.365} C_VEL
LIN {X 0,Y 375.048,Z 973.615,A -85,B 0,C 180,E1 -358.581,E2 -358.581} C_VEL
LIN {X 0,Y 375.048,Z 1022.694,A -85,B 0,C 180,E1 -358.581,E2 -358.581} C_VEL
LIN {X 0,Y 353.26,Z 1022.694,A -85,B 0,C 180,E1 -358.212,E2 -358.212} C_VEL
LIN {X 0,Y 351.272,Z 1020.694,A -85,B 0,C 180,E1 -358.176,E2 -358.176} C_VEL
LIN {X 0,Y 351.272,Z 1011.577,A -85,B 0,C 180,E1 -358.176,E2 -358.176} C_VEL
LIN {X 0,Y 347.855,Z 1010.408,A -85,B 0,C 180,E1 -358.373,E2 -358.373} C_VEL
LIN {X 0,Y 330.977,Z 1032.743,A -85,B 0,C 180,E1 -359.374,E2 -359.374} C_VEL
LIN {X 0,Y 316.963,Z 1049.362,A -85,B 0,C 180,E1 -360.304,E2 -360.304} C_VEL
LIN {X 0,Y 302.049,Z 1065.454,A -85,B 0,C 180,E1 -361.391,E2 -361.391} C_VEL
LIN {X 0,Y 283.334,Z 1083.786,A -85,B 0,C 180,E1 -362.934,E2 -362.934} C_VEL
LIN {X 0,Y 263.887,Z 1100.63,A -85,B 0,C 180,E1 -364.79,E2 -364.79} C_VEL
LIN {X 0,Y 246.656,Z 1114.206,A -85,B 0,C 180,E1 -366.708,E2 -366.708} C_VEL
LIN {X 0,Y 228.735,Z 1127.106,A -85,B 0,C 180,E1 -369.054,E2 -369.054} C_VEL
LIN {X 0,Y 206.021,Z 1141.857,A -85,B 0,C 180,E1 -372.71,E2 -372.71} C_VEL
LIN {X 0,Y 186.787,Z 1153.026,A -85,B 0,C 180,E1 -376.629,E2 -376.629} C_VEL
LIN {X 0,Y 169.382,Z 1162.317,A -85,B 0,C 180,E1 -381.145,E2 -381.145} C_VEL
LIN {X 0,Y 149.535,Z 1172.087,A -85,B 0,C 180,E1 -388.041,E2 -388.041} C_VEL
LIN {X 0,Y 133.48,Z 1179.311,A -85,B 0,C 180,E1 -396.003,E2 -396.003} C_VEL
LIN {X 0,Y 121.789,Z 1184.451,A -85,B 0,C 180,E1 -404.419,E2 -404.419} C_VEL
LIN {X 0,Y 112.829,Z 1188.482,A -85,B 0,C 180,E1 -414.206,E2 -414.206} C_VEL
LIN {X 0,Y 106.809,Z 1191.545,A -85,B 0,C 180,E1 -425.677,E2 -425.677} C_VEL
LIN {X 0,Y 104.251,Z 1193.462,A -85,B 0,C 180,E1 -438.045,E2 -438.045} C_VEL
LIN {X 0,Y 104.043,Z 1193.974,A -85,B 0,C 180,E1 -446.696,E2 -446.696} C_VEL
LIN {X 0,Y 104.043,Z 1193.968,A -85,B 0,C 180,E1 -453.307,E2 -453.307} C_VEL
LIN {X 0,Y 104.267,Z 1193.417,A -85,B 0,C 180,E1 -462.18,E2 -462.18} C_VEL
LIN {X 0,Y 106.807,Z 1191.518,A -85,B 0,C 180,E1 -474.326,E2 -474.326} C_VEL
LIN {X 0,Y 112.478,Z 1188.613,A -85,B 0,C 180,E1 -485.298,E2 -485.298} C_VEL
LIN {X 0,Y 121.296,Z 1184.618,A -85,B 0,C 180,E1 -495.149,E2 -495.149} C_VEL
LIN {X 0,Y 132.869,Z 1179.514,A -85,B 0,C 180,E1 -503.632,E2 -503.632} C_VEL
LIN {X 0,Y 149.534,Z 1172.009,A -85,B 0,C 180,E1 -511.963,E2 -511.963} C_VEL
LIN {X 0,Y 168.58,Z 1162.628,A -85,B 0,C 180,E1 -518.624,E2 -518.624} C_VEL
LIN {X 0,Y 185.935,Z 1153.378,A -85,B 0,C 180,E1 -523.18,E2 -523.18} C_VEL
LIN {X 0,Y 203.348,Z 1143.307,A -85,B 0,C 180,E1 -526.802,E2 -526.802} C_VEL
LIN {X 0,Y 225.111,Z 1129.475,A -85,B 0,C 180,E1 -530.425,E2 -530.425} C_VEL
LIN {X 0,Y 244.76,Z 1115.436,A -85,B 0,C 180,E1 -533.07,E2 -533.07} C_VEL
LIN {X 0,Y 261.959,Z 1101.978,A -85,B 0,C 180,E1 -535.018,E2 -535.018} C_VEL
LIN {X 0,Y 279.424,Z 1087.008,A -85,B 0,C 180,E1 -536.723,E2 -536.723} C_VEL
LIN {X 0,Y 300.191,Z 1067.087,A -85,B 0,C 180,E1 -538.473,E2 -538.473} C_VEL
LIN {X 0,Y 315.471,Z 1050.713,A -85,B 0,C 180,E1 -539.605,E2 -539.605} C_VEL
LIN {X 0,Y 329.978,Z 1033.597,A -85,B 0,C 180,E1 -540.575,E2 -540.575} C_VEL
LIN {X 0,Y 346.414,Z 1012.063,A -85,B 0,C 180,E1 -541.555,E2 -541.555} C_VEL
LIN {X 0,Y 348.409,Z 1009.131,A -85,B 0,C 180,E1 -541.673,E2 -541.673} C_VEL
LIN {X 0,Y 331.323,Z 1031.864,A -85,B 0,C 180,E1 -542.677,E2 -542.677} C_VEL
LIN {X 0,Y 316.601,Z 1049.26,A -85,B 0,C 180,E1 -543.639,E2 -543.639} C_VEL
LIN {X 0,Y 301.195,Z 1065.742,A -85,B 0,C 180,E1 -544.761,E2 -544.761} C_VEL
LIN {X 0,Y 281.709,Z 1084.481,A -85,B 0,C 180,E1 -546.374,E2 -546.374} C_VEL
LIN {X 0,Y 263.603,Z 1099.904,A -85,B 0,C 180,E1 -548.105,E2 -548.105} C_VEL
LIN {X 0,Y 246.704,Z 1112.993,A -85,B 0,C 180,E1 -549.978,E2 -549.978} C_VEL
LIN {X 0,Y 228.14,Z 1126.066,A -85,B 0,C 180,E1 -552.401,E2 -552.401} C_VEL
LIN {X 0,Y 205.919,Z 1140.006,A -85,B 0,C 180,E1 -555.964,E2 -555.964} C_VEL
LIN {X 0,Y 187.867,Z 1150.128,A -85,B 0,C 180,E1 -559.601,E2 -559.601} C_VEL
LIN {X 0,Y 170.693,Z 1158.905,A -85,B 0,C 180,E1 -563.961,E2 -563.961} C_VEL
LIN {X 0,Y 150.897,Z 1168.106,A -85,B 0,C 180,E1 -570.679,E2 -570.679} C_VEL
LIN {X 0,Y 135.022,Z 1174.726,A -85,B 0,C 180,E1 -578.282,E2 -578.282} C_VEL
LIN {X 0,Y 123.225,Z 1179.406,A -85,B 0,C 180,E1 -586.392,E2 -586.392} C_VEL
LIN {X 0,Y 113.666,Z 1183.157,A -85,B 0,C 180,E1 -596.344,E2 -596.344} C_VEL
LIN {X 0,Y 106.66,Z 1186.153,A -85,B 0,C 180,E1 -609.704,E2 -609.704} C_VEL
LIN {X 0,Y 104.351,Z 1187.365,A -85,B 0,C 180,E1 -621.735,E2 -621.735} C_VEL
LIN {X 0,Y 104.101,Z 1187.642,A -85,B 0,C 180,E1 -631.1,E2 -631.1} C_VEL
LIN {X 0,Y 104.623,Z 1187.25,A -85,B 0,C 180,E1 -641.018,E2 -641.018} C_VEL
LIN {X 0,Y 108.038,Z 1185.498,A -85,B 0,C 180,E1 -654.029,E2 -654.029} C_VEL
LIN {X 0,Y 114.721,Z 1182.767,A -85,B 0,C 180,E1 -665.115,E2 -665.115} C_VEL
LIN {X 0,Y 124.692,Z 1178.895,A -85,B 0,C 180,E1 -674.881,E2 -674.881} C_VEL
LIN {X 0,Y 140.018,Z 1172.853,A -85,B 0,C 180,E1 -684.495,E2 -684.495} C_VEL
LIN {X 0,Y 157.894,Z 1165.011,A -85,B 0,C 180,E1 -692.055,E2 -692.055} C_VEL
LIN {X 0,Y 173.804,Z 1157.475,A -85,B 0,C 180,E1 -696.992,E2 -696.992} C_VEL
LIN {X 0,Y 192.018,Z 1148.046,A -85,B 0,C 180,E1 -701.387,E2 -701.387} C_VEL
LIN {X 0,Y 213.8,Z 1135.401,A -85,B 0,C 180,E1 -705.481,E2 -705.481} C_VEL
LIN {X 0,Y 231.866,Z 1123.689,A -85,B 0,C 180,E1 -708.205,E2 -708.205} C_VEL
LIN {X 0,Y 248.508,Z 1111.854,A -85,B 0,C 180,E1 -710.317,E2 -710.317} C_VEL
LIN {X 0,Y 267.343,Z 1097.131,A -85,B 0,C 180,E1 -712.352,E2 -712.352} C_VEL
LIN {X 0,Y 287.512,Z 1079.352,A -85,B 0,C 180,E1 -714.212,E2 -714.212} C_VEL
LIN {X 0,Y 303.052,Z 1064.131,A -85,B 0,C 180,E1 -715.458,E2 -715.458} C_VEL
LIN {X 0,Y 318.039,Z 1047.985,A -85,B 0,C 180,E1 -716.537,E2 -716.537} C_VEL
LIN {X 0,Y 335.241,Z 1027.435,A -85,B 0,C 180,E1 -717.639,E2 -717.639} C_VEL
LIN {X 0,Y 347.855,Z 1010.408,A -85,B 0,C 180,E1 -718.373,E2 -718.373} C_VEL
LIN {X 0,Y 350.166,Z 1011.83,A -85,B 0,C 180,E1 -718.784,E2 -718.784} C_VEL
LIN {X 0,Y 350.166,Z 1052.626,A -85,B 0,C 180,E1 -718.784,E2 -718.784} C_VEL
LIN {X 0,Y 329.192,Z 1052.626,A -85,B 0,C 180,E1 -718.229,E2 -718.229} C_VEL
LIN {X 0,Y 327.218,Z 1050.626,A -85,B 0,C 180,E1 -718.174,E2 -718.174} C_VEL
LIN {X 0,Y 327.218,Z 1042.563,A -85,B 0,C 180,E1 -718.174,E2 -718.174} C_VEL
LIN {X 0,Y 323.906,Z 1041.251,A -85,B 0,C 180,E1 -718.378,E2 -718.378} C_VEL
LIN {X 0,Y 305.469,Z 1061.54,A -85,B 0,C 180,E1 -719.562,E2 -719.562} C_VEL
LIN {X 0,Y 288.988,Z 1077.843,A -85,B 0,C 180,E1 -720.764,E2 -720.764} C_VEL
LIN {X 0,Y 271.173,Z 1093.838,A -85,B 0,C 180,E1 -722.251,E2 -722.251} C_VEL
LIN {X 0,Y 248.717,Z 1111.783,A -85,B 0,C 180,E1 -724.449,E2 -724.449} C_VEL
LIN {X 0,Y 230.489,Z 1124.83,A -85,B 0,C 180,E1 -726.584,E2 -726.584} C_VEL
LIN {X 0,Y 212.633,Z 1136.488,A -85,B 0,C 180,E1 -729.075,E2 -729.075} C_VEL
LIN {X 0,Y 190.753,Z 1149.456,A -85,B 0,C 180,E1 -732.852,E2 -732.852} C_VEL
LIN {X 0,Y 169.87,Z 1160.381,A -85,B 0,C 180,E1 -737.534,E2 -737.534} C_VEL
LIN {X 0,Y 152.71,Z 1168.605,A -85,B 0,C 180,E1 -742.603,E2 -742.603} C_VEL
LIN {X 0,Y 134.121,Z 1176.867,A -85,B 0,C 180,E1 -750.144,E2 -750.144} C_VEL
LIN {X 0,Y 117.578,Z 1183.597,A -85,B 0,C 180,E1 -760.264,E2 -760.264} C_VEL
LIN {X 0,Y 106.997,Z 1187.886,A -85,B 0,C 180,E1 -770.548,E2 -770.548} C_VEL
LIN {X 0,Y 100.319,Z 1190.803,A -85,B 0,C 180,E1 -781.419,E2 -781.419} C_VEL
LIN {X 0,Y 96.913,Z 1192.661,A -85,B 0,C 180,E1 -792.592,E2 -792.592} C_VEL
LIN {X 0,Y 96.073,Z 1193.545,A -85,B 0,C 180,E1 -802.225,E2 -802.225} C_VEL
LIN {X 0,Y 96.069,Z 1193.841,A -85,B 0,C 180,E1 -810.598,E2 -810.598} C_VEL
LIN {X 0,Y 96.115,Z 1193.459,A -85,B 0,C 180,E1 -819.583,E2 -819.583} C_VEL
LIN {X 0,Y 98.181,Z 1191.968,A -85,B 0,C 180,E1 -832.769,E2 -832.769} C_VEL
LIN {X 0,Y 105.118,Z 1188.658,A -85,B 0,C 180,E1 -846.963,E2 -846.963} C_VEL
LIN {X 0,Y 115.008,Z 1184.576,A -85,B 0,C 180,E1 -857.647,E2 -857.647} C_VEL
LIN {X 0,Y 127.407,Z 1179.519,A -85,B 0,C 180,E1 -866.294,E2 -866.294} C_VEL
LIN {X 0,Y 143.496,Z 1172.691,A -85,B 0,C 180,E1 -874.011,E2 -874.011} C_VEL
LIN {X 0,Y 164.853,Z 1162.778,A -85,B 0,C 180,E1 -881.12,E2 -881.12} C_VEL
LIN {X 0,Y 182.786,Z 1153.579,A -85,B 0,C 180,E1 -885.521,E2 -885.521} C_VEL
LIN {X 0,Y 200.674,Z 1143.564,A -85,B 0,C 180,E1 -888.987,E2 -888.987} C_VEL
LIN {X 0,Y 221.979,Z 1130.466,A -85,B 0,C 180,E1 -892.296,E2 -892.296} C_VEL
LIN {X 0,Y 242.925,Z 1115.866,A -85,B 0,C 180,E1 -894.925,E2 -894.925} C_VEL
LIN {X 0,Y 260.387,Z 1102.473,A -85,B 0,C 180,E1 -896.757,E2 -896.757} C_VEL
LIN {X 0,Y 278.082,Z 1087.57,A -85,B 0,C 180,E1 -898.356,E2 -898.356} C_VEL
LIN {X 0,Y 299.195,Z 1067.68,A -85,B 0,C 180,E1 -900,E2 -900} C_VEL
LIN {X 0,Y 315.185,Z 1050.756,A -85,B 0,C 180,E1 -901.091,E2 -901.091} C_VEL
LIN {X 0,Y 324.426,Z 1040.241,A -85,B 0,C 180,E1 -901.667,E2 -901.667} C_VEL
LIN {X 0,Y 305.844,Z 1060.738,A -85,B 0,C 180,E1 -902.855,E2 -902.855} C_VEL
LIN {X 0,Y 289.678,Z 1076.673,A -85,B 0,C 180,E1 -904.017,E2 -904.017} C_VEL
LIN {X 0,Y 272.199,Z 1092.28,A -85,B 0,C 180,E1 -905.451,E2 -905.451} C_VEL
LIN {X 0,Y 250.107,Z 1109.854,A -85,B 0,C 180,E1 -907.581,E2 -907.581} C_VEL
LIN {X 0,Y 231.311,Z 1123.119,A -85,B 0,C 180,E1 -909.745,E2 -909.745} C_VEL
LIN {X 0,Y 212.856,Z 1134.912,A -85,B 0,C 180,E1 -912.292,E2 -912.292} C_VEL
LIN {X 0,Y 190.358,Z 1147.763,A -85,B 0,C 180,E1 -916.164,E2 -916.164} C_VEL
LIN {X 0,Y 170.815,Z 1157.589,A -85,B 0,C 180,E1 -920.515,E2 -920.515} C_VEL
LIN {X 0,Y 153.878,Z 1165.309,A -85,B 0,C 180,E1 -925.416,E2 -925.416} C_VEL
LIN {X 0,Y 134.775,Z 1173.266,A -85,B 0,C 180,E1 -933.034,E2 -933.034} C_VEL
LIN {X 0,Y 119.066,Z 1179.069,A -85,B 0,C 180,E1 -942.353,E2 -942.353} C_VEL
LIN {X 0,Y 108.594,Z 1182.804,A -85,B 0,C 180,E1 -951.908,E2 -951.908} C_VEL
LIN {X 0,Y 101.207,Z 1185.489,A -85,B 0,C 180,E1 -962.969,E2 -962.969} C_VEL
LIN {X 0,Y 97.317,Z 1187.092,A -85,B 0,C 180,E1 -974.505,E2 -974.505} C_VEL
LIN {X 0,Y 96.202,Z 1187.712,A -85,B 0,C 180,E1 -984.033,E2 -984.033} C_VEL
LIN {X 0,Y 96.112,Z 1187.846,A -85,B 0,C 180,E1 -992.384,E2 -992.384} C_VEL
LIN {X 0,Y 96.895,Z 1187.372,A -85,B 0,C 180,E1 -1003.121,E2 -1003.121} C_VEL
LIN {X 0,Y 100.905,Z 1185.642,A -85,B 0,C 180,E1 -1016.48,E2 -1016.48} C_VEL
LIN {X 0,Y 108.112,Z 1183.019,A -85,B 0,C 180,E1 -1027.617,E2 -1027.617} C_VEL
LIN {X 0,Y 118.996,Z 1179.148,A -85,B 0,C 180,E1 -1037.681,E2 -1037.681} C_VEL
LIN {X 0,Y 135.553,Z 1173.042,A -85,B 0,C 180,E1 -1047.42,E2 -1047.42} C_VEL
LIN {X 0,Y 153.798,Z 1165.439,A -85,B 0,C 180,E1 -1054.643,E2 -1054.643} C_VEL
LIN {X 0,Y 170.74,Z 1157.732,A -85,B 0,C 180,E1 -1059.548,E2 -1059.548} C_VEL
LIN {X 0,Y 189.615,Z 1148.266,A -85,B 0,C 180,E1 -1063.771,E2 -1063.771} C_VEL
LIN {X 0,Y 212.793,Z 1135.104,A -85,B 0,C 180,E1 -1067.78,E2 -1067.78} C_VEL
LIN {X 0,Y 231.257,Z 1123.334,A -85,B 0,C 180,E1 -1070.328,E2 -1070.328} C_VEL
LIN {X 0,Y 249.157,Z 1110.749,A -85,B 0,C 180,E1 -1072.398,E2 -1072.398} C_VEL
LIN {X 0,Y 271.195,Z 1093.401,A -85,B 0,C 180,E1 -1074.539,E2 -1074.539} C_VEL
LIN {X 0,Y 288.672,Z 1077.896,A -85,B 0,C 180,E1 -1075.982,E2 -1075.982} C_VEL
LIN {X 0,Y 304.344,Z 1062.575,A -85,B 0,C 180,E1 -1077.121,E2 -1077.121} C_VEL
LIN {X 0,Y 321.115,Z 1044.459,A -85,B 0,C 180,E1 -1078.208,E2 -1078.208} C_VEL
LIN {X 0,Y 323.906,Z 1041.251,A -85,B 0,C 180,E1 -1078.378,E2 -1078.378} C_VEL
LIN {X 0,Y 316.758,Z 1049.597,A -85,B 0,C 180,E1 -1078.648,E2 -1078.648} C_VEL
LIN {X 0,Y 308.189,Z 1058.825,A -85,B 0,C 180,E1 -1078.619,E2 -1078.619} C_VEL
LIN {X 0,Y 297.201,Z 1069.811,A -85,B 0,C 180,E1 -1078.186,E2 -1078.186} C_VEL
LIN {X 0,Y 291.373,Z 1075.265,A -85,B 0,C 180,E1 -1077.823,E2 -1077.823} C_VEL
LIN {X 0,Y 274.454,Z 1090.352,A -85,B 0,C 180,E1 -1076.577,E2 -1076.577} C_VEL
LIN {X 0,Y 255.939,Z 1105.289,A -85,B 0,C 180,E1 -1075.004,E2 -1075.004} C_VEL
LIN {X 0,Y 233.825,Z 1121.104,A -85,B 0,C 180,E1 -1072.776,E2 -1072.776} C_VEL
LIN {X 0,Y 214.934,Z 1133.117,A -85,B 0,C 180,E1 -1070.476,E2 -1070.476} C_VEL
LIN {X 0,Y 196.45,Z 1143.734,A -85,B 0,C 180,E1 -1067.746,E2 -1067.746} C_VEL
LIN {X 0,Y 174.1,Z 1155.224,A -85,B 0,C 180,E1 -1063.554,E2 -1063.554} C_VEL
LIN {X 0,Y 153.715,Z 1164.321,A -85,B 0,C 180,E1 -1058.461,E2 -1058.461} C_VEL
LIN {X 0,Y 137.066,Z 1171.018,A -85,B 0,C 180,E1 -1052.868,E2 -1052.868} C_VEL
LIN {X 0,Y 119.961,Z 1177.295,A -85,B 0,C 180,E1 -1044.767,E2 -1044.767} C_VEL
LIN {X 0,Y 104.156,Z 1182.513,A -85,B 0,C 180,E1 -1032.966,E2 -1032.966} C_VEL
LIN {X 0,Y 94.935,Z 1185.466,A -85,B 0,C 180,E1 -1021.068,E2 -1021.068} C_VEL
LIN {X 0,Y 89.979,Z 1187.181,A -85,B 0,C 180,E1 -1008.798,E2 -1008.798} C_VEL
LIN {X 0,Y 88.302,Z 1187.929,A -85,B 0,C 180,E1 -997.808,E2 -997.808} C_VEL
LIN {X 0,Y 88.109,Z 1188.106,A -85,B 0,C 180,E1 -988.048,E2 -988.048} C_VEL
LIN {X 0,Y 88.963,Z 1187.658,A -85,B 0,C 180,E1 -976.347,E2 -976.347} C_VEL
LIN {X 0,Y 93.416,Z 1185.955,A -85,B 0,C 180,E1 -961.902,E2 -961.902} C_VEL
LIN {X 0,Y 101.79,Z 1183.21,A -85,B 0,C 180,E1 -949.584,E2 -949.584} C_VEL
LIN {X 0,Y 113.678,Z 1179.325,A -85,B 0,C 180,E1 -939.282,E2 -939.282} C_VEL
LIN {X 0,Y 131.184,Z 1173.257,A -85,B 0,C 180,E1 -929.667,E2 -929.667} C_VEL
LIN {X 0,Y 150.515,Z 1165.569,A -85,B 0,C 180,E1 -922.572,E2 -922.572} C_VEL
LIN {X 0,Y 168.095,Z 1157.849,A -85,B 0,C 180,E1 -917.873,E2 -917.873} C_VEL
LIN {X 0,Y 188.357,Z 1147.959,A -85,B 0,C 180,E1 -913.724,E2 -913.724} C_VEL
LIN {X 0,Y 211.479,Z 1135.043,A -85,B 0,C 180,E1 -910.075,E2 -910.075} C_VEL
LIN {X 0,Y 230.062,Z 1123.39,A -85,B 0,C 180,E1 -907.725,E2 -907.725} C_VEL
LIN {X 0,Y 248.502,Z 1110.6,A -85,B 0,C 180,E1 -905.773,E2 -905.773} C_VEL
LIN {X 0,Y 271.545,Z 1092.573,A -85,B 0,C 180,E1 -903.733,E2 -903.733} C_VEL
LIN {X 0,Y 289.221,Z 1076.975,A -85,B 0,C 180,E1 -902.405,E2 -902.405} C_VEL
LIN {X 0,Y 300.285,Z 1066.368,A -85,B 0,C 180,E1 -901.663,E2 -901.663} C_VEL
LIN {X 0,Y 278.969,Z 1086.412,A -85,B 0,C 180,E1 -900.159,E2 -900.159} C_VEL
LIN {X 0,Y 260.047,Z 1102.183,A -85,B 0,C 180,E1 -898.605,E2 -898.605} C_VEL
LIN {X 0,Y 242.325,Z 1115.583,A -85,B 0,C 180,E1 -896.906,E2 -896.906} C_VEL
LIN {X 0,Y 220.046,Z 1130.778,A -85,B 0,C 180,E1 -894.344,E2 -894.344} C_VEL
LIN {X 0,Y 198.919,Z 1143.468,A -85,B 0,C 180,E1 -891.327,E2 -891.327} C_VEL
LIN {X 0,Y 180.854,Z 1153.31,A -85,B 0,C 180,E1 -888.119,E2 -888.119} C_VEL
LIN {X 0,Y 161.45,Z 1162.927,A -85,B 0,C 180,E1 -883.728,E2 -883.728} C_VEL
LIN {X 0,Y 139.216,Z 1172.743,A -85,B 0,C 180,E1 -876.829,E2 -876.829} C_VEL
LIN {X 0,Y 122.936,Z 1179.257,A -85,B 0,C 180,E1 -869.559,E2 -869.559} C_VEL
LIN {X 0,Y 109.537,Z 1184.316,A -85,B 0,C 180,E1 -860.888,E2 -860.888} C_VEL
LIN {X 0,Y 98.092,Z 1188.605,A -85,B 0,C 180,E1 -849.198,E2 -849.198} C_VEL
LIN {X 0,Y 90.105,Z 1191.934,A -85,B 0,C 180,E1 -832.92,E2 -832.92} C_VEL
LIN {X 0,Y 88.124,Z 1193.236,A -85,B 0,C 180,E1 -819.8,E2 -819.8} C_VEL
LIN {X 0,Y 88.072,Z 1193.594,A -85,B 0,C 180,E1 -810.652,E2 -810.652} C_VEL
LIN {X 0,Y 88.09,Z 1193.297,A -85,B 0,C 180,E1 -801.516,E2 -801.516} C_VEL
LIN {X 0,Y 89.436,Z 1192.26,A -85,B 0,C 180,E1 -789.724,E2 -789.724} C_VEL
LIN {X 0,Y 94.124,Z 1190.158,A -85,B 0,C 180,E1 -777.059,E2 -777.059} C_VEL
LIN {X 0,Y 104.61,Z 1186.27,A -85,B 0,C 180,E1 -763.415,E2 -763.415} C_VEL
LIN {X 0,Y 120.199,Z 1180.386,A -85,B 0,C 180,E1 -751.955,E2 -751.955} C_VEL
LIN {X 0,Y 136.116,Z 1174.087,A -85,B 0,C 180,E1 -744.376,E2 -744.376} C_VEL
LIN {X 0,Y 153.81,Z 1166.515,A -85,B 0,C 180,E1 -738.361,E2 -738.361} C_VEL
LIN {X 0,Y 177.26,Z 1155.323,A -85,B 0,C 180,E1 -732.622,E2 -732.622} C_VEL
LIN {X 0,Y 197.367,Z 1144.488,A -85,B 0,C 180,E1 -728.932,E2 -728.932} C_VEL
LIN {X 0,Y 216.221,Z 1133.283,A -85,B 0,C 180,E1 -726.163,E2 -726.163} C_VEL
LIN {X 0,Y 238.417,Z 1118.642,A -85,B 0,C 180,E1 -723.517,E2 -723.517} C_VEL
LIN {X 0,Y 259.054,Z 1103.199,A -85,B 0,C 180,E1 -721.494,E2 -721.494} C_VEL
LIN {X 0,Y 275.964,Z 1089.249,A -85,B 0,C 180,E1 -720.085,E2 -720.085} C_VEL
LIN {X 0,Y 294.029,Z 1072.842,A -85,B 0,C 180,E1 -718.769,E2 -718.769} C_VEL
LIN {X 0,Y 299.655,Z 1067.317,A -85,B 0,C 180,E1 -718.372,E2 -718.372} C_VEL
LIN {X 0,Y 291.373,Z 1075.265,A -85,B 0,C 180,E1 -717.823,E2 -717.823} C_VEL
LIN {X 0,Y 286.501,Z 1079.797,A -85,B 0,C 180,E1 -717.672,E2 -717.672} C_VEL
LIN {X 0,Y 280.713,Z 1085.033,A -85,B 0,C 180,E1 -717.852,E2 -717.852} C_VEL
LIN {X 0,Y 264.701,Z 1098.438,A -85,B 0,C 180,E1 -719.187,E2 -719.187} C_VEL
LIN {X 0,Y 244.994,Z 1113.369,A -85,B 0,C 180,E1 -720.844,E2 -720.844} C_VEL
LIN {X 0,Y 226.223,Z 1126.226,A -85,B 0,C 180,E1 -722.71,E2 -722.71} C_VEL
LIN {X 0,Y 202.922,Z 1140.526,A -85,B 0,C 180,E1 -725.545,E2 -725.545} C_VEL
LIN {X 0,Y 181.333,Z 1152.14,A -85,B 0,C 180,E1 -728.882,E2 -728.882} C_VEL
LIN {X 0,Y 162.858,Z 1161.105,A -85,B 0,C 180,E1 -732.531,E2 -732.531} C_VEL
LIN {X 0,Y 141.729,Z 1170.363,A -85,B 0,C 180,E1 -738.085,E2 -738.085} C_VEL
LIN {X 0,Y 120.821,Z 1178.374,A -85,B 0,C 180,E1 -746.016,E2 -746.016} C_VEL
LIN {X 0,Y 105.719,Z 1183.675,A -85,B 0,C 180,E1 -754.632,E2 -754.632} C_VEL
LIN {X 0,Y 93.708,Z 1187.711,A -85,B 0,C 180,E1 -765.235,E2 -765.235} C_VEL
LIN {X 0,Y 84.892,Z 1190.782,A -85,B 0,C 180,E1 -778.787,E2 -778.787} C_VEL
LIN {X 0,Y 80.512,Z 1192.754,A -85,B 0,C 180,E1 -794.884,E2 -794.884} C_VEL
LIN {X 0,Y 80.048,Z 1193.256,A -85,B 0,C 180,E1 -806.421,E2 -806.421} C_VEL
LIN {X 0,Y 80.048,Z 1193.25,A -85,B 0,C 180,E1 -813.582,E2 -813.582} C_VEL
LIN {X 0,Y 80.512,Z 1192.737,A -85,B 0,C 180,E1 -825.119,E2 -825.119} C_VEL
LIN {X 0,Y 84.89,Z 1190.753,A -85,B 0,C 180,E1 -841.217,E2 -841.217} C_VEL
LIN {X 0,Y 93.219,Z 1187.839,A -85,B 0,C 180,E1 -854.204,E2 -854.204} C_VEL
LIN {X 0,Y 105.081,Z 1183.838,A -85,B 0,C 180,E1 -864.918,E2 -864.918} C_VEL
LIN {X 0,Y 119.63,Z 1178.728,A -85,B 0,C 180,E1 -873.423,E2 -873.423} C_VEL
LIN {X 0,Y 140.266,Z 1170.899,A -85,B 0,C 180,E1 -881.459,E2 -881.459} C_VEL
LIN {X 0,Y 161.961,Z 1161.406,A -85,B 0,C 180,E1 -887.274,E2 -887.274} C_VEL
LIN {X 0,Y 180.233,Z 1152.571,A -85,B 0,C 180,E1 -890.932,E2 -890.932} C_VEL
LIN {X 0,Y 200.049,Z 1141.967,A -85,B 0,C 180,E1 -894.067,E2 -894.067} C_VEL
LIN {X 0,Y 224.265,Z 1127.339,A -85,B 0,C 180,E1 -897.085,E2 -897.085} C_VEL
LIN {X 0,Y 243.833,Z 1113.995,A -85,B 0,C 180,E1 -899.06,E2 -899.06} C_VEL
LIN {X 0,Y 261.985,Z 1100.324,A -85,B 0,C 180,E1 -900.614,E2 -900.614} C_VEL
LIN {X 0,Y 276.039,Z 1088.732,A -85,B 0,C 180,E1 -901.661,E2 -901.661} C_VEL
LIN {X 0,Y 259.307,Z 1102.276,A -85,B 0,C 180,E1 -902.919,E2 -902.919} C_VEL
LIN {X 0,Y 240.726,Z 1115.896,A -85,B 0,C 180,E1 -904.535,E2 -904.535} C_VEL
LIN {X 0,Y 216.627,Z 1131.503,A -85,B 0,C 180,E1 -907.08,E2 -907.08} C_VEL
LIN {X 0,Y 197.716,Z 1142.312,A -85,B 0,C 180,E1 -909.546,E2 -909.546} C_VEL
LIN {X 0,Y 178.754,Z 1152.051,A -85,B 0,C 180,E1 -912.601,E2 -912.601} C_VEL
LIN {X 0,Y 156.097,Z 1162.389,A -85,B 0,C 180,E1 -917.364,E2 -917.364} C_VEL
LIN {X 0,Y 135.974,Z 1170.286,A -85,B 0,C 180,E1 -923.192,E2 -923.192} C_VEL
LIN {X 0,Y 119.039,Z 1176.234,A -85,B 0,C 180,E1 -930.097,E2 -930.097} C_VEL
LIN {X 0,Y 102.378,Z 1181.56,A -85,B 0,C 180,E1 -940.376,E2 -940.376} C_VEL
LIN {X 0,Y 88.851,Z 1185.461,A -85,B 0,C 180,E1 -954.974,E2 -954.974} C_VEL
LIN {X 0,Y 82.564,Z 1187.342,A -85,B 0,C 180,E1 -968.695,E2 -968.695} C_VEL
LIN {X 0,Y 80.418,Z 1188.149,A -85,B 0,C 180,E1 -980.697,E2 -980.697} C_VEL
LIN {X 0,Y 80.113,Z 1188.383,A -85,B 0,C 180,E1 -991.429,E2 -991.429} C_VEL
LIN {X 0,Y 81.008,Z 1187.997,A -85,B 0,C 180,E1 -1004.29,E2 -1004.29} C_VEL
LIN {X 0,Y 86.268,Z 1186.251,A -85,B 0,C 180,E1 -1020.66,E2 -1020.66} C_VEL
LIN {X 0,Y 95.634,Z 1183.524,A -85,B 0,C 180,E1 -1033.632,E2 -1033.632} C_VEL
LIN {X 0,Y 108.581,Z 1179.654,A -85,B 0,C 180,E1 -1044.129,E2 -1044.129} C_VEL
LIN {X 0,Y 127.228,Z 1173.62,A -85,B 0,C 180,E1 -1053.625,E2 -1053.625} C_VEL
LIN {X 0,Y 147.475,Z 1165.953,A -85,B 0,C 180,E1 -1060.459,E2 -1060.459} C_VEL
LIN {X 0,Y 165.685,Z 1158.248,A -85,B 0,C 180,E1 -1064.918,E2 -1064.918} C_VEL
LIN {X 0,Y 185.597,Z 1148.821,A -85,B 0,C 180,E1 -1068.663,E2 -1068.663} C_VEL
LIN {X 0,Y 209.922,Z 1135.636,A -85,B 0,C 180,E1 -1072.184,E2 -1072.184} C_VEL
LIN {X 0,Y 229.067,Z 1123.873,A -85,B 0,C 180,E1 -1074.389,E2 -1074.389} C_VEL
LIN {X 0,Y 247.52,Z 1111.298,A -85,B 0,C 180,E1 -1076.168,E2 -1076.168} C_VEL
LIN {X 0,Y 270.13,Z 1093.976,A -85,B 0,C 180,E1 -1077.996,E2 -1077.996} C_VEL
LIN {X 0,Y 275.507,Z 1089.443,A -85,B 0,C 180,E1 -1078.388,E2 -1078.388} C_VEL
LIN {X 0,Y 264.701,Z 1098.438,A -85,B 0,C 180,E1 -1079.187,E2 -1079.187} C_VEL
LIN {X 0,Y 258.61,Z 1103.169,A -85,B 0,C 180,E1 -1079.435,E2 -1079.435} C_VEL
LIN {X 0,Y 241.473,Z 1115.711,A -85,B 0,C 180,E1 -1079.357,E2 -1079.357} C_VEL
LIN {X 0,Y 236.083,Z 1119.397,A -85,B 0,C 180,E1 -1079.636,E2 -1079.636} C_VEL
LIN {X 0,Y 213.263,Z 1133.811,A -85,B 0,C 180,E1 -1081.881,E2 -1081.881} C_VEL
LIN {X 0,Y 193.516,Z 1145.005,A -85,B 0,C 180,E1 -1084.288,E2 -1084.288} C_VEL
LIN {X 0,Y 169.632,Z 1157.083,A -85,B 0,C 180,E1 -1088.009,E2 -1088.009} C_VEL
LIN {X 0,Y 147.549,Z 1166.721,A -85,B 0,C 180,E1 -1092.627,E2 -1092.627} C_VEL
LIN {X 0,Y 129.208,Z 1173.879,A -85,B 0,C 180,E1 -1097.859,E2 -1097.859} C_VEL
LIN {X 0,Y 109.913,Z 1180.662,A -85,B 0,C 180,E1 -1105.765,E2 -1105.765} C_VEL
LIN {X 0,Y 91.447,Z 1186.435,A -85,B 0,C 180,E1 -1118.074,E2 -1118.074} C_VEL
LIN {X 0,Y 80.232,Z 1189.793,A -85,B 0,C 180,E1 -1131.458,E2 -1131.458} C_VEL
LIN {X 0,Y 74.083,Z 1191.83,A -85,B 0,C 180,E1 -1146.117,E2 -1146.117} C_VEL
LIN {X 0,Y 72.118,Z 1192.825,A -85,B 0,C 180,E1 -1160.425,E2 -1160.425} C_VEL
LIN {X 0,Y 72.076,Z 1193.1,A -85,B 0,C 180,E1 -1170.797,E2 -1170.797} C_VEL
LIN {X 0,Y 72.228,Z 1192.736,A -85,B 0,C 180,E1 -1181.986,E2 -1181.986} C_VEL
LIN {X 0,Y 75.858,Z 1191.251,A -85,B 0,C 180,E1 -1199.546,E2 -1199.546} C_VEL
LIN {X 0,Y 86.508,Z 1187.872,A -85,B 0,C 180,E1 -1217.004,E2 -1217.004} C_VEL
LIN {X 0,Y 99.806,Z 1183.794,A -85,B 0,C 180,E1 -1228.383,E2 -1228.383} C_VEL
LIN {X 0,Y 115.314,Z 1178.731,A -85,B 0,C 180,E1 -1236.8,E2 -1236.8} C_VEL
LIN {X 0,Y 134.338,Z 1171.904,A -85,B 0,C 180,E1 -1243.773,E2 -1243.773} C_VEL
LIN {X 0,Y 158.465,Z 1161.974,A -85,B 0,C 180,E1 -1249.845,E2 -1249.845} C_VEL
LIN {X 0,Y 178.142,Z 1152.774,A -85,B 0,C 180,E1 -1253.453,E2 -1253.453} C_VEL
LIN {X 0,Y 197.404,Z 1142.751,A -85,B 0,C 180,E1 -1256.235,E2 -1256.235} C_VEL
LIN {X 0,Y 221.013,Z 1129,A -85,B 0,C 180,E1 -1258.939,E2 -1258.939} C_VEL
LIN {X 0,Y 242.752,Z 1114.482,A -85,B 0,C 180,E1 -1260.944,E2 -1260.944} C_VEL
LIN {X 0,Y 251.635,Z 1108.19,A -85,B 0,C 180,E1 -1261.655,E2 -1261.655} C_VEL
LIN {X 0,Y 230.012,Z 1122.929,A -85,B 0,C 180,E1 -1263.489,E2 -1263.489} C_VEL
LIN {X 0,Y 211.892,Z 1134.026,A -85,B 0,C 180,E1 -1265.329,E2 -1265.329} C_VEL
LIN {X 0,Y 191.757,Z 1145.101,A -85,B 0,C 180,E1 -1267.809,E2 -1267.809} C_VEL
LIN {X 0,Y 166.523,Z 1157.182,A -85,B 0,C 180,E1 -1271.836,E2 -1271.836} C_VEL
LIN {X 0,Y 146.729,Z 1165.399,A -85,B 0,C 180,E1 -1276.086,E2 -1276.086} C_VEL
LIN {X 0,Y 127.885,Z 1172.322,A -85,B 0,C 180,E1 -1281.56,E2 -1281.56} C_VEL
LIN {X 0,Y 105.347,Z 1179.467,A -85,B 0,C 180,E1 -1291.469,E2 -1291.469} C_VEL
LIN {X 0,Y 90.497,Z 1183.568,A -85,B 0,C 180,E1 -1302.244,E2 -1302.244} C_VEL
LIN {X 0,Y 80.174,Z 1186.248,A -85,B 0,C 180,E1 -1314.991,E2 -1314.991} C_VEL
LIN {X 0,Y 74.008,Z 1187.906,A -85,B 0,C 180,E1 -1330.258,E2 -1330.258} C_VEL
LIN {X 0,Y 72.219,Z 1188.496,A -85,B 0,C 180,E1 -1343.639,E2 -1343.639} C_VEL
LIN {X 0,Y 72.134,Z 1188.576,A -85,B 0,C 180,E1 -1353.595,E2 -1353.595} C_VEL
LIN {X 0,Y 73.487,Z 1188.12,A -85,B 0,C 180,E1 -1367.416,E2 -1367.416} C_VEL
LIN {X 0,Y 79.739,Z 1186.396,A -85,B 0,C 180,E1 -1384.35,E2 -1384.35} C_VEL
LIN {X 0,Y 89.893,Z 1183.77,A -85,B 0,C 180,E1 -1397.272,E2 -1397.272} C_VEL
LIN {X 0,Y 103.961,Z 1179.908,A -85,B 0,C 180,E1 -1407.817,E2 -1407.817} C_VEL
LIN {X 0,Y 123.775,Z 1173.875,A -85,B 0,C 180,E1 -1417.057,E2 -1417.057} C_VEL
LIN {X 0,Y 145.104,Z 1166.138,A -85,B 0,C 180,E1 -1423.589,E2 -1423.589} C_VEL
LIN {X 0,Y 163.727,Z 1158.507,A -85,B 0,C 180,E1 -1427.715,E2 -1427.715} C_VEL
LIN {X 0,Y 184.15,Z 1149.082,A -85,B 0,C 180,E1 -1431.185,E2 -1431.185} C_VEL
LIN {X 0,Y 208.961,Z 1135.902,A -85,B 0,C 180,E1 -1434.423,E2 -1434.423} C_VEL
LIN {X 0,Y 228.41,Z 1124.143,A -85,B 0,C 180,E1 -1436.442,E2 -1436.442} C_VEL
LIN {X 0,Y 247.108,Z 1111.57,A -85,B 0,C 180,E1 -1438.067,E2 -1438.067} C_VEL
LIN {X 0,Y 251.025,Z 1108.836,A -85,B 0,C 180,E1 -1438.402,E2 -1438.402} C_VEL
LIN {X 0,Y 236.083,Z 1119.397,A -85,B 0,C 180,E1 -1439.636,E2 -1439.636} C_VEL
LIN {X 0,Y 229.67,Z 1123.632,A -85,B 0,C 180,E1 -1439.956,E2 -1439.956} C_VEL
LIN {X 0,Y 211.468,Z 1134.569,A -85,B 0,C 180,E1 -1439.993,E2 -1439.993} C_VEL
LIN {X 0,Y 205.846,Z 1137.82,A -85,B 0,C 180,E1 -1440.36,E2 -1440.36} C_VEL
LIN {X 0,Y 181.276,Z 1150.754,A -85,B 0,C 180,E1 -1443.302,E2 -1443.302} C_VEL
LIN {X 0,Y 160.994,Z 1160.158,A -85,B 0,C 180,E1 -1446.442,E2 -1446.442} C_VEL
LIN {X 0,Y 141.311,Z 1168.282,A -85,B 0,C 180,E1 -1450.421,E2 -1450.421} C_VEL
LIN {X 0,Y 117.271,Z 1176.964,A -85,B 0,C 180,E1 -1457.363,E2 -1457.363} C_VEL
LIN {X 0,Y 97.849,Z 1182.961,A -85,B 0,C 180,E1 -1466.066,E2 -1466.066} C_VEL
LIN {X 0,Y 83.319,Z 1187.028,A -85,B 0,C 180,E1 -1476.485,E2 -1476.485} C_VEL
LIN {X 0,Y 72.11,Z 1190.028,A -85,B 0,C 180,E1 -1490.372,E2 -1490.372} C_VEL
LIN {X 0,Y 65.583,Z 1191.953,A -85,B 0,C 180,E1 -1507.597,E2 -1507.597} C_VEL
LIN {X 0,Y 64.068,Z 1192.683,A -85,B 0,C 180,E1 -1522.83,E2 -1522.83} C_VEL
LIN {X 0,Y 64.071,Z 1192.829,A -85,B 0,C 180,E1 -1531.79,E2 -1531.79} C_VEL
LIN {X 0,Y 64.393,Z 1192.458,A -85,B 0,C 180,E1 -1544.387,E2 -1544.387} C_VEL
LIN {X 0,Y 69.36,Z 1190.852,A -85,B 0,C 180,E1 -1564.211,E2 -1564.211} C_VEL
LIN {X 0,Y 81.481,Z 1187.491,A -85,B 0,C 180,E1 -1581.757,E2 -1581.757} C_VEL
LIN {X 0,Y 96.416,Z 1183.316,A -85,B 0,C 180,E1 -1593.111,E2 -1593.111} C_VEL
LIN {X 0,Y 113.932,Z 1177.939,A -85,B 0,C 180,E1 -1601.412,E2 -1601.412} C_VEL
LIN {X 0,Y 136.743,Z 1170.005,A -85,B 0,C 180,E1 -1608.475,E2 -1608.475} C_VEL
LIN {X 0,Y 159.093,Z 1160.875,A -85,B 0,C 180,E1 -1613.227,E2 -1613.227} C_VEL
LIN {X 0,Y 178.351,Z 1152.036,A -85,B 0,C 180,E1 -1616.303,E2 -1616.303} C_VEL
LIN {X 0,Y 200.007,Z 1140.899,A -85,B 0,C 180,E1 -1619.017,E2 -1619.017} C_VEL
LIN {X 0,Y 225.049,Z 1126.13,A -85,B 0,C 180,E1 -1621.481,E2 -1621.481} C_VEL
LIN {X 0,Y 227.069,Z 1124.835,A -85,B 0,C 180,E1 -1621.658,E2 -1621.658} C_VEL
LIN {X 0,Y 205.406,Z 1137.676,A -85,B 0,C 180,E1 -1623.703,E2 -1623.703} C_VEL
LIN {X 0,Y 181.178,Z 1150.092,A -85,B 0,C 180,E1 -1626.593,E2 -1626.593} C_VEL
LIN {X 0,Y 161.271,Z 1159.024,A -85,B 0,C 180,E1 -1629.665,E2 -1629.665} C_VEL
LIN {X 0,Y 141.034,Z 1167.033,A -85,B 0,C 180,E1 -1633.762,E2 -1633.762} C_VEL
LIN {X 0,Y 116.632,Z 1175.272,A -85,B 0,C 180,E1 -1640.858,E2 -1640.858} C_VEL
LIN {X 0,Y 98.368,Z 1180.488,A -85,B 0,C 180,E1 -1649.051,E2 -1649.051} C_VEL
LIN {X 0,Y 83.318,Z 1184.278,A -85,B 0,C 180,E1 -1659.819,E2 -1659.819} C_VEL
LIN {X 0,Y 70.319,Z 1187.344,A -85,B 0,C 180,E1 -1677.292,E2 -1677.292} C_VEL
LIN {X 0,Y 64.807,Z 1188.608,A -85,B 0,C 180,E1 -1696.617,E2 -1696.617} C_VEL
LIN {X 0,Y 64.12,Z 1188.911,A -85,B 0,C 180,E1 -1709.998,E2 -1709.998} C_VEL
LIN {X 0,Y 64.912,Z 1188.597,A -85,B 0,C 180,E1 -1724.266,E2 -1724.266} C_VEL
LIN {X 0,Y 71.443,Z 1187.076,A -85,B 0,C 180,E1 -1745.015,E2 -1745.015} C_VEL
LIN {X 0,Y 83.979,Z 1184.158,A -85,B 0,C 180,E1 -1760.873,E2 -1760.873} C_VEL
LIN {X 0,Y 99.057,Z 1180.36,A -85,B 0,C 180,E1 -1771.42,E2 -1771.42} C_VEL
LIN {X 0,Y 118.253,Z 1174.869,A -85,B 0,C 180,E1 -1779.806,E2 -1779.806} C_VEL
LIN {X 0,Y 142.135,Z 1166.719,A -85,B 0,C 180,E1 -1786.576,E2 -1786.576} C_VEL
LIN {X 0,Y 162.168,Z 1158.766,A -85,B 0,C 180,E1 -1790.573,E2 -1790.573} C_VEL
LIN {X 0,Y 182.934,Z 1149.405,A -85,B 0,C 180,E1 -1793.724,E2 -1793.724} C_VEL
LIN {X 0,Y 208.542,Z 1136.041,A -85,B 0,C 180,E1 -1796.702,E2 -1796.702} C_VEL
LIN {X 0,Y 226.605,Z 1125.322,A -85,B 0,C 180,E1 -1798.392,E2 -1798.392} C_VEL
LIN {X 0,Y 205.846,Z 1137.82,A -85,B 0,C 180,E1 -1800.36,E2 -1800.36} C_VEL
LIN {X 0,Y 199.193,Z 1141.525,A -85,B 0,C 180,E1 -1800.786,E2 -1800.786} C_VEL
LIN {X 0,Y 180.141,Z 1150.931,A -85,B 0,C 180,E1 -1800.983,E2 -1800.983} C_VEL
LIN {X 0,Y 174.265,Z 1153.677,A -85,B 0,C 180,E1 -1801.458,E2 -1801.458} C_VEL
LIN {X 0,Y 147.671,Z 1165.1,A -85,B 0,C 180,E1 -1805.545,E2 -1805.545} C_VEL
LIN {X 0,Y 126.911,Z 1172.725,A -85,B 0,C 180,E1 -1810.002,E2 -1810.002} C_VEL
LIN {X 0,Y 107.15,Z 1179.078,A -85,B 0,C 180,E1 -1816.027,E2 -1816.027} C_VEL
LIN {X 0,Y 85.895,Z 1185.063,A -85,B 0,C 180,E1 -1826.323,E2 -1826.323} C_VEL
LIN {X 0,Y 68.595,Z 1189.16,A -85,B 0,C 180,E1 -1841.981,E2 -1841.981} C_VEL
LIN {X 0,Y 59.759,Z 1191.248,A -85,B 0,C 180,E1 -1858.758,E2 -1858.758} C_VEL
LIN {X 0,Y 56.294,Z 1192.298,A -85,B 0,C 180,E1 -1876.652,E2 -1876.652} C_VEL
LIN {X 0,Y 56.079,Z 1192.611,A -85,B 0,C 180,E1 -1888.981,E2 -1888.981} C_VEL
LIN {X 0,Y 56.178,Z 1192.347,A -85,B 0,C 180,E1 -1901.293,E2 -1901.293} C_VEL
LIN {X 0,Y 58.873,Z 1191.455,A -85,B 0,C 180,E1 -1918.397,E2 -1918.397} C_VEL
LIN {X 0,Y 66.978,Z 1189.494,A -85,B 0,C 180,E1 -1935.774,E2 -1935.774} C_VEL
LIN {X 0,Y 80.043,Z 1186.384,A -85,B 0,C 180,E1 -1949.537,E2 -1949.537} C_VEL
LIN {X 0,Y 99.48,Z 1181.319,A -85,B 0,C 180,E1 -1960.877,E2 -1960.877} C_VEL
LIN {X 0,Y 122.317,Z 1174.21,A -85,B 0,C 180,E1 -1968.8,E2 -1968.8} C_VEL
LIN {X 0,Y 143.004,Z 1166.776,A -85,B 0,C 180,E1 -1973.577,E2 -1973.577} C_VEL
LIN {X 0,Y 164.542,Z 1157.954,A -85,B 0,C 180,E1 -1977.213,E2 -1977.213} C_VEL
LIN {X 0,Y 190.986,Z 1145.372,A -85,B 0,C 180,E1 -1980.519,E2 -1980.519} C_VEL
LIN {X 0,Y 202.322,Z 1139.437,A -85,B 0,C 180,E1 -1981.654,E2 -1981.654} C_VEL
LIN {X 0,Y 178.932,Z 1151.039,A -85,B 0,C 180,E1 -1984.166,E2 -1984.166} C_VEL
LIN {X 0,Y 159.133,Z 1159.681,A -85,B 0,C 180,E1 -1986.894,E2 -1986.894} C_VEL
LIN {X 0,Y 135.589,Z 1168.668,A -85,B 0,C 180,E1 -1991.246,E2 -1991.246} C_VEL
LIN {X 0,Y 112.206,Z 1176.019,A -85,B 0,C 180,E1 -1997.541,E2 -1997.541} C_VEL
LIN {X 0,Y 93.842,Z 1180.941,A -85,B 0,C 180,E1 -2005.084,E2 -2005.084} C_VEL
LIN {X 0,Y 76.974,Z 1184.836,A -85,B 0,C 180,E1 -2016.352,E2 -2016.352} C_VEL
LIN {X 0,Y 62.363,Z 1187.784,A -85,B 0,C 180,E1 -2035.862,E2 -2035.862} C_VEL
LIN {X 0,Y 56.865,Z 1188.875,A -85,B 0,C 180,E1 -2055.747,E2 -2055.747} C_VEL
LIN {X 0,Y 56.121,Z 1189.147,A -85,B 0,C 180,E1 -2071.019,E2 -2071.019} C_VEL
LIN {X 0,Y 57.28,Z 1188.828,A -85,B 0,C 180,E1 -2087.26,E2 -2087.26} C_VEL
LIN {X 0,Y 65.399,Z 1187.221,A -85,B 0,C 180,E1 -2109.948,E2 -2109.948} C_VEL
LIN {X 0,Y 78.941,Z 1184.436,A -85,B 0,C 180,E1 -2125.414,E2 -2125.414} C_VEL
LIN {X 0,Y 95.386,Z 1180.615,A -85,B 0,C 180,E1 -2135.776,E2 -2135.776} C_VEL
LIN {X 0,Y 115.658,Z 1175.124,A -85,B 0,C 180,E1 -2143.655,E2 -2143.655} C_VEL
LIN {X 0,Y 140.192,Z 1167.07,A -85,B 0,C 180,E1 -2149.811,E2 -2149.811} C_VEL
LIN {X 0,Y 160.061,Z 1159.421,A -85,B 0,C 180,E1 -2153.331,E2 -2153.331} C_VEL
LIN {X 0,Y 180.395,Z 1150.502,A -85,B 0,C 180,E1 -2156.092,E2 -2156.092} C_VEL
LIN {X 0,Y 201.871,Z 1139.822,A -85,B 0,C 180,E1 -2158.397,E2 -2158.397} C_VEL
LIN {X 0,Y 178.996,Z 1151.432,A -85,B 0,C 180,E1 -2160.869,E2 -2160.869} C_VEL
LIN {X 0,Y 174.265,Z 1153.677,A -85,B 0,C 180,E1 -2161.458,E2 -2161.458} C_VEL
LIN {X 0,Y 167.353,Z 1156.828,A -85,B 0,C 180,E1 -2162.021,E2 -2162.021} C_VEL
LIN {X 0,Y 147.649,Z 1164.693,A -85,B 0,C 180,E1 -2162.489,E2 -2162.489} C_VEL
LIN {X 0,Y 141.614,Z 1166.876,A -85,B 0,C 180,E1 -2163.158,E2 -2163.158} C_VEL
LIN {X 0,Y 119.115,Z 1174.65,A -85,B 0,C 180,E1 -2167.719,E2 -2167.719} C_VEL
LIN {X 0,Y 93.528,Z 1181.987,A -85,B 0,C 180,E1 -2175.817,E2 -2175.817} C_VEL
LIN {X 0,Y 75.368,Z 1186.342,A -85,B 0,C 180,E1 -2185.564,E2 -2185.564} C_VEL
LIN {X 0,Y 60.874,Z 1189.394,A -85,B 0,C 180,E1 -2199.47,E2 -2199.47} C_VEL
LIN {X 0,Y 51.142,Z 1191.373,A -85,B 0,C 180,E1 -2219.45,E2 -2219.45} C_VEL
LIN {X 0,Y 48.12,Z 1192.186,A -85,B 0,C 180,E1 -2240.434,E2 -2240.434} C_VEL
LIN {X 0,Y 48.068,Z 1192.334,A -85,B 0,C 180,E1 -2252.387,E2 -2252.387} C_VEL
LIN {X 0,Y 48.81,Z 1191.956,A -85,B 0,C 180,E1 -2269.135,E2 -2269.135} C_VEL
LIN {X 0,Y 56.466,Z 1190.34,A -85,B 0,C 180,E1 -2293.681,E2 -2293.681} C_VEL
LIN {X 0,Y 72.343,Z 1186.973,A -85,B 0,C 180,E1 -2312.202,E2 -2312.202} C_VEL
LIN {X 0,Y 90.07,Z 1182.796,A -85,B 0,C 180,E1 -2322.692,E2 -2322.692} C_VEL
LIN {X 0,Y 109.727,Z 1177.417,A -85,B 0,C 180,E1 -2329.788,E2 -2329.788} C_VEL
LIN {X 0,Y 135.511,Z 1169.053,A -85,B 0,C 180,E1 -2335.768,E2 -2335.768} C_VEL
LIN {X 0,Y 158.989,Z 1159.927,A -85,B 0,C 180,E1 -2339.466,E2 -2339.466} C_VEL
LIN {X 0,Y 177.056,Z 1151.967,A -85,B 0,C 180,E1 -2341.677,E2 -2341.677} C_VEL
LIN {X 0,Y 155.426,Z 1161.129,A -85,B 0,C 180,E1 -2344.326,E2 -2344.326} C_VEL
LIN {X 0,Y 128.534,Z 1170.727,A -85,B 0,C 180,E1 -2348.899,E2 -2348.899} C_VEL
LIN {X 0,Y 108.186,Z 1176.767,A -85,B 0,C 180,E1 -2353.964,E2 -2353.964} C_VEL
LIN {X 0,Y 88.971,Z 1181.592,A -85,B 0,C 180,E1 -2361.124,E2 -2361.124} C_VEL
LIN {X 0,Y 68.152,Z 1185.941,A -85,B 0,C 180,E1 -2374.753,E2 -2374.753} C_VEL
LIN {X 0,Y 54.028,Z 1188.284,A -85,B 0,C 180,E1 -2394.988,E2 -2394.988} C_VEL
LIN {X 0,Y 48.797,Z 1189.162,A -85,B 0,C 180,E1 -2415.763,E2 -2415.763} C_VEL
LIN {X 0,Y 48.125,Z 1189.394,A -85,B 0,C 180,E1 -2431.188,E2 -2431.188} C_VEL
LIN {X 0,Y 49.621,Z 1189.077,A -85,B 0,C 180,E1 -2450.03,E2 -2450.03} C_VEL
LIN {X 0,Y 59.368,Z 1187.473,A -85,B 0,C 180,E1 -2475.018,E2 -2475.018} C_VEL
LIN {X 0,Y 75.332,Z 1184.538,A -85,B 0,C 180,E1 -2491.161,E2 -2491.161} C_VEL
LIN {X 0,Y 93.163,Z 1180.672,A -85,B 0,C 180,E1 -2500.811,E2 -2500.811} C_VEL
LIN {X 0,Y 116.369,Z 1174.64,A -85,B 0,C 180,E1 -2508.38,E2 -2508.38} C_VEL
LIN {X 0,Y 140.884,Z 1166.64,A -85,B 0,C 180,E1 -2513.507,E2 -2513.507} C_VEL
LIN {X 0,Y 161.271,Z 1158.889,A -85,B 0,C 180,E1 -2516.543,E2 -2516.543} C_VEL
LIN {X 0,Y 176.759,Z 1152.243,A -85,B 0,C 180,E1 -2518.409,E2 -2518.409} C_VEL
LIN {X 0,Y 154.014,Z 1162.133,A -85,B 0,C 180,E1 -2521.228,E2 -2521.228} C_VEL
LIN {X 0,Y 141.614,Z 1166.876,A -85,B 0,C 180,E1 -2523.158,E2 -2523.158} C_VEL
LIN {X 0,Y 134.53,Z 1169.482,A -85,B 0,C 180,E1 -2523.965,E2 -2523.965} C_VEL
LIN {X 0,Y 113.787,Z 1175.829,A -85,B 0,C 180,E1 -2524.965,E2 -2524.965} C_VEL
LIN {X 0,Y 108.177,Z 1177.333,A -85,B 0,C 180,E1 -2525.917,E2 -2525.917} C_VEL
LIN {X 0,Y 87.932,Z 1182.596,A -85,B 0,C 180,E1 -2532.072,E2 -2532.072} C_VEL
LIN {X 0,Y 68.841,Z 1186.762,A -85,B 0,C 180,E1 -2541.638,E2 -2541.638} C_VEL
LIN {X 0,Y 49.636,Z 1190.283,A -85,B 0,C 180,E1 -2561.816,E2 -2561.816} C_VEL
LIN {X 0,Y 41.006,Z 1191.74,A -85,B 0,C 180,E1 -2588.549,E2 -2588.549} C_VEL
LIN {X 0,Y 40.066,Z 1192.093,A -85,B 0,C 180,E1 -2607.142,E2 -2607.142} C_VEL
LIN {X 0,Y 40.129,Z 1191.957,A -85,B 0,C 180,E1 -2620.048,E2 -2620.048} C_VEL
LIN {X 0,Y 43.993,Z 1191.152,A -85,B 0,C 180,E1 -2645.092,E2 -2645.092} C_VEL
LIN {X 0,Y 55.281,Z 1189.226,A -85,B 0,C 180,E1 -2666.31,E2 -2666.31} C_VEL
LIN {X 0,Y 71.317,Z 1186.206,A -85,B 0,C 180,E1 -2679.947,E2 -2679.947} C_VEL
LIN {X 0,Y 90.676,Z 1181.885,A -85,B 0,C 180,E1 -2688.937,E2 -2688.937} C_VEL
LIN {X 0,Y 116.281,Z 1174.942,A -85,B 0,C 180,E1 -2695.932,E2 -2695.932} C_VEL
LIN {X 0,Y 139.985,Z 1167.022,A -85,B 0,C 180,E1 -2700.071,E2 -2700.071} C_VEL
LIN {X 0,Y 151.683,Z 1162.722,A -85,B 0,C 180,E1 -2701.684,E2 -2701.684} C_VEL
LIN {X 0,Y 126.211,Z 1171.382,A -85,B 0,C 180,E1 -2705.455,E2 -2705.455} C_VEL
LIN {X 0,Y 105.556,Z 1177.271,A -85,B 0,C 180,E1 -2709.884,E2 -2709.884} C_VEL
LIN {X 0,Y 84.572,Z 1182.245,A -85,B 0,C 180,E1 -2716.73,E2 -2716.73} C_VEL
LIN {X 0,Y 60.836,Z 1186.62,A -85,B 0,C 180,E1 -2731.274,E2 -2731.274} C_VEL
LIN {X 0,Y 47.094,Z 1188.597,A -85,B 0,C 180,E1 -2750.433,E2 -2750.433} C_VEL
LIN {X 0,Y 41.042,Z 1189.411,A -85,B 0,C 180,E1 -2772.999,E2 -2772.999} C_VEL
LIN {X 0,Y 40.128,Z 1189.641,A -85,B 0,C 180,E1 -2791.425,E2 -2791.425} C_VEL
LIN {X 0,Y 42.115,Z 1189.327,A -85,B 0,C 180,E1 -2813.801,E2 -2813.801} C_VEL
LIN {X 0,Y 53.9,Z 1187.726,A -85,B 0,C 180,E1 -2841.177,E2 -2841.177} C_VEL
LIN {X 0,Y 71.726,Z 1184.792,A -85,B 0,C 180,E1 -2856.929,E2 -2856.929} C_VEL
LIN {X 0,Y 90.785,Z 1180.927,A -85,B 0,C 180,E1 -2865.738,E2 -2865.738} C_VEL
LIN {X 0,Y 114.989,Z 1174.895,A -85,B 0,C 180,E1 -2872.419,E2 -2872.419} C_VEL
LIN {X 0,Y 140.19,Z 1166.898,A -85,B 0,C 180,E1 -2876.869,E2 -2876.869} C_VEL
LIN {X 0,Y 151.535,Z 1162.91,A -85,B 0,C 180,E1 -2878.389,E2 -2878.389} C_VEL
LIN {X 0,Y 126.073,Z 1171.89,A -85,B 0,C 180,E1 -2882.169,E2 -2882.169} C_VEL
LIN {X 0,Y 108.177,Z 1177.333,A -85,B 0,C 180,E1 -2885.917,E2 -2885.917} C_VEL
LIN {X 0,Y 101.005,Z 1179.272,A -85,B 0,C 180,E1 -2887.176,E2 -2887.176} C_VEL
LIN {X 0,Y 79.963,Z 1183.924,A -85,B 0,C 180,E1 -2889.33,E2 -2889.33} C_VEL
LIN {X 0,Y 74.373,Z 1184.972,A -85,B 0,C 180,E1 -2890.991,E2 -2890.991} C_VEL
LIN {X 0,Y 54.303,Z 1188.512,A -85,B 0,C 180,E1 -2902.986,E2 -2902.986} C_VEL
LIN {X 0,Y 40.109,Z 1190.562,A -85,B 0,C 180,E1 -2921.598,E2 -2921.598} C_VEL
LIN {X 0,Y 32.858,Z 1191.574,A -85,B 0,C 180,E1 -2948.587,E2 -2948.587} C_VEL
LIN {X 0,Y 32.095,Z 1191.884,A -85,B 0,C 180,E1 -2970.004,E2 -2970.004} C_VEL
LIN {X 0,Y 32.858,Z 1191.567,A -85,B 0,C 180,E1 -2991.422,E2 -2991.422} C_VEL
LIN {X 0,Y 40.11,Z 1190.541,A -85,B 0,C 180,E1 -3018.409,E2 -3018.409} C_VEL
LIN {X 0,Y 55.117,Z 1188.355,A -85,B 0,C 180,E1 -3037.703,E2 -3037.703} C_VEL
LIN {X 0,Y 78.067,Z 1184.229,A -85,B 0,C 180,E1 -3050.485,E2 -3050.485} C_VEL
LIN {X 0,Y 103.078,Z 1178.222,A -85,B 0,C 180,E1 -3057.623,E2 -3057.623} C_VEL
LIN {X 0,Y 124.026,Z 1172.163,A -85,B 0,C 180,E1 -3061.386,E2 -3061.386} C_VEL
LIN {X 0,Y 125.693,Z 1171.64,A -85,B 0,C 180,E1 -3061.701,E2 -3061.701} C_VEL
LIN {X 0,Y 104.455,Z 1177.528,A -85,B 0,C 180,E1 -3065.411,E2 -3065.411} C_VEL
LIN {X 0,Y 82.577,Z 1182.501,A -85,B 0,C 180,E1 -3071.242,E2 -3071.242} C_VEL
LIN {X 0,Y 57.01,Z 1186.874,A -85,B 0,C 180,E1 -3084.21,E2 -3084.21} C_VEL
LIN {X 0,Y 41.147,Z 1188.849,A -85,B 0,C 180,E1 -3103.192,E2 -3103.192} C_VEL
LIN {X 0,Y 33.192,Z 1189.678,A -85,B 0,C 180,E1 -3130.644,E2 -3130.644} C_VEL
LIN {X 0,Y 32.131,Z 1189.888,A -85,B 0,C 180,E1 -3151.779,E2 -3151.779} C_VEL
LIN {X 0,Y 34.527,Z 1189.594,A -85,B 0,C 180,E1 -3177.599,E2 -3177.599} C_VEL
LIN {X 0,Y 48.453,Z 1188.085,A -85,B 0,C 180,E1 -3207.783,E2 -3207.783} C_VEL
LIN {X 0,Y 68.492,Z 1185.12,A -85,B 0,C 180,E1 -3223.024,E2 -3223.024} C_VEL
LIN {X 0,Y 88.167,Z 1181.381,A -85,B 0,C 180,E1 -3230.616,E2 -3230.616} C_VEL
LIN {X 0,Y 110.348,Z 1176.118,A -85,B 0,C 180,E1 -3235.843,E2 -3235.843} C_VEL
LIN {X 0,Y 125.595,Z 1171.767,A -85,B 0,C 180,E1 -3238.387,E2 -3238.387} C_VEL
LIN {X 0,Y 103.899,Z 1178.077,A -85,B 0,C 180,E1 -3242.206,E2 -3242.206} C_VEL
LIN {X 0,Y 78.997,Z 1184.074,A -85,B 0,C 180,E1 -3249.169,E2 -3249.169} C_VEL
LIN {X 0,Y 74.373,Z 1184.972,A -85,B 0,C 180,E1 -3250.991,E2 -3250.991} C_VEL
LIN {X 0,Y 67.275,Z 1186.225,A -85,B 0,C 180,E1 -3253.334,E2 -3253.334} C_VEL
LIN {X 0,Y 46.431,Z 1189.164,A -85,B 0,C 180,E1 -3259.291,E2 -3259.291} C_VEL
LIN {X 0,Y 41.177,Z 1189.711,A -85,B 0,C 180,E1 -3263.362,E2 -3263.362} C_VEL
LIN {X 0,Y 26.246,Z 1191.256,A -85,B 0,C 180,E1 -3296.944,E2 -3296.944} C_VEL
LIN {X 0,Y 24.069,Z 1191.623,A -85,B 0,C 180,E1 -3327.624,E2 -3327.624} C_VEL
LIN {X 0,Y 24.517,Z 1191.43,A -85,B 0,C 180,E1 -3349.048,E2 -3349.048} C_VEL
LIN {X 0,Y 32.423,Z 1190.591,A -85,B 0,C 180,E1 -3383.308,E2 -3383.308} C_VEL
LIN {X 0,Y 48.18,Z 1188.7,A -85,B 0,C 180,E1 -3403.109,E2 -3403.109} C_VEL
LIN {X 0,Y 68.393,Z 1185.519,A -85,B 0,C 180,E1 -3413.809,E2 -3413.809} C_VEL
LIN {X 0,Y 90.991,Z 1180.93,A -85,B 0,C 180,E1 -3420.073,E2 -3420.073} C_VEL
LIN {X 0,Y 99.288,Z 1178.952,A -85,B 0,C 180,E1 -3421.669,E2 -3421.669} C_VEL
LIN {X 0,Y 71.76,Z 1184.488,A -85,B 0,C 180,E1 -3428.382,E2 -3428.382} C_VEL
LIN {X 0,Y 51.049,Z 1187.502,A -85,B 0,C 180,E1 -3438.264,E2 -3438.264} C_VEL
LIN {X 0,Y 34.648,Z 1189.225,A -85,B 0,C 180,E1 -3456.09,E2 -3456.09} C_VEL
LIN {X 0,Y 25.432,Z 1189.946,A -85,B 0,C 180,E1 -3486.843,E2 -3486.843} C_VEL
LIN {X 0,Y 24.159,Z 1190.113,A -85,B 0,C 180,E1 -3514.743,E2 -3514.743} C_VEL
LIN {X 0,Y 28.563,Z 1189.809,A -85,B 0,C 180,E1 -3549.052,E2 -3549.052} C_VEL
LIN {X 0,Y 47.152,Z 1188.018,A -85,B 0,C 180,E1 -3578.906,E2 -3578.906} C_VEL
LIN {X 0,Y 67.009,Z 1185.301,A -85,B 0,C 180,E1 -3589.996,E2 -3589.996} C_VEL
LIN {X 0,Y 88.181,Z 1181.438,A -85,B 0,C 180,E1 -3596.202,E2 -3596.202} C_VEL
LIN {X 0,Y 99.025,Z 1179.097,A -85,B 0,C 180,E1 -3598.381,E2 -3598.381} C_VEL
LIN {X 0,Y 71.28,Z 1185.057,A -85,B 0,C 180,E1 -3605.175,E2 -3605.175} C_VEL
LIN {X 0,Y 50.729,Z 1188.379,A -85,B 0,C 180,E1 -3615.039,E2 -3615.039} C_VEL
LIN {X 0,Y 41.177,Z 1189.711,A -85,B 0,C 180,E1 -3623.362,E2 -3623.362} C_VEL
LIN {X 0,Y 34.775,Z 1190.307,A -85,B 0,C 180,E1 -3629.95,E2 -3629.95} C_VEL
LIN {X 0,Y 23.919,Z 1191.038,A -85,B 0,C 180,E1 -3643.659,E2 -3643.659} C_VEL
LIN {X 0,Y 16.504,Z 1191.283,A -85,B 0,C 180,E1 -3672.569,E2 -3672.569} C_VEL
LIN {X 0,Y 16.076,Z 1191.346,A -85,B 0,C 180,E1 -3682.349,E2 -3682.349} C_VEL
LIN {X 0,Y 16.207,Z 1191.29,A -85,B 0,C 180,E1 -3704.294,E2 -3704.294} C_VEL
LIN {X 0,Y 25.883,Z 1190.564,A -85,B 0,C 180,E1 -3752.697,E2 -3752.697} C_VEL
LIN {X 0,Y 45.394,Z 1188.579,A -85,B 0,C 180,E1 -3772.414,E2 -3772.414} C_VEL
LIN {X 0,Y 66.997,Z 1185.43,A -85,B 0,C 180,E1 -3780.596,E2 -3780.596} C_VEL
LIN {X 0,Y 71.448,Z 1184.678,A -85,B 0,C 180,E1 -3781.694,E2 -3781.694} C_VEL
LIN {X 0,Y 49.593,Z 1187.701,A -85,B 0,C 180,E1 -3788.901,E2 -3788.901} C_VEL
LIN {X 0,Y 30.567,Z 1189.477,A -85,B 0,C 180,E1 -3803.653,E2 -3803.653} C_VEL
LIN {X 0,Y 18.301,Z 1190.195,A -85,B 0,C 180,E1 -3836.875,E2 -3836.875} C_VEL
LIN {X 0,Y 16.144,Z 1190.382,A -85,B 0,C 180,E1 -3873.543,E2 -3873.543} C_VEL
LIN {X 0,Y 21.527,Z 1190.094,A -85,B 0,C 180,E1 -3917.993,E2 -3917.993} C_VEL
LIN {X 0,Y 42.07,Z 1188.591,A -85,B 0,C 180,E1 -3947.005,E2 -3947.005} C_VEL
LIN {X 0,Y 65.093,Z 1185.707,A -85,B 0,C 180,E1 -3956.776,E2 -3956.776} C_VEL
LIN {X 0,Y 71.016,Z 1184.799,A -85,B 0,C 180,E1 -3958.414,E2 -3958.414} C_VEL
LIN {X 0,Y 49.229,Z 1188.122,A -85,B 0,C 180,E1 -3965.624,E2 -3965.624} C_VEL
LIN {X 0,Y 30.797,Z 1190.129,A -85,B 0,C 180,E1 -3979.701,E2 -3979.701} C_VEL
LIN {X 0,Y 18.199,Z 1191.1,A -85,B 0,C 180,E1 -4012.826,E2 -4012.826} C_VEL
LIN {X 0,Y 16.076,Z 1191.346,A -85,B 0,C 180,E1 -4042.349,E2 -4042.349} C_VEL
LIN {X 0,Y 15.871,Z 1191.389,A -85,B 0,C 180,E1 -4061.979,E2 -4061.979} C_VEL
LIN {X 0,Y 16.36,Z 1191.214,A -85,B 0,C 180,E1 -4087.731,E2 -4087.731} C_VEL
LIN {X 0,Y 26.004,Z 1190.122,A -85,B 0,C 180,E1 -4132.28,E2 -4132.28} C_VEL
LIN {X 0,Y 30.657,Z 1189.729,A -85,B 0,C 180,E1 -4136.854,E2 -4136.854} C_VEL
LIN {X 0,Y 41.277,Z 1188.779,A -85,B 0,C 180,E1 -4141.744,E2 -4141.744} C_VEL
LIN {X 0,Y 17.205,Z 1190.337,A -85,B 0,C 180,E1 -4161.574,E2 -4161.574} C_VEL
LIN {X 0,Y 8.172,Z 1190.622,A -85,B 0,C 180,E1 -4222.957,E2 -4222.957} C_VEL
LIN {X 0,Y 13.579,Z 1190.422,A -85,B 0,C 180,E1 -4288.973,E2 -4288.973} C_VEL
LIN {X 0,Y 31.186,Z 1189.566,A -85,B 0,C 180,E1 -4313.639,E2 -4313.639} C_VEL
LIN {X 0,Y 41.01,Z 1188.847,A -85,B 0,C 180,E1 -4318.354,E2 -4318.354} C_VEL
LIN {X 0,Y 16.85,Z 1190.702,A -85,B 0,C 180,E1 -4338.325,E2 -4338.325} C_VEL
LIN {X 0,Y 8.08,Z 1191.142,A -85,B 0,C 180,E1 -4410.015,E2 -4410.015} C_VEL
LIN {X 0,Y 16.854,Z 1190.695,A -85,B 0,C 180,E1 -4481.68,E2 -4481.68} C_VEL
LIN {X 0,Y 30.657,Z 1189.729,A -85,B 0,C 180,E1 -4496.854,E2 -4496.854} C_VEL
LIN {X 0,Y 29.045,Z 1189.823,A -85,B 0,C 180,E1 -4498.499,E2 -4498.499} C_VEL
LIN {X 0,Y 19.854,Z 1190.418,A -85,B 0,C 180,E1 -4499.324,E2 -4499.324} C_VEL
LIN {X 0,Y 1.112,Z 1190.901,A -85,B 0,C 180,E1 -4492.478,E2 -4492.478} C_VEL
LIN {X 0,Y 0.337,Z 1190.89,A -85,B 0,C 180,E1 -4325.753,E2 -4325.753} C_VEL
